(* IEC 61131-3 sources: TA/Tests/RetainTest/OLD/Array test (part 5) *)

    ARRAY_ARRAY_REAL_AUTO[4][0] := ARRAY_ARRAY_REAL_AUTO[4][0] + 1;
    ARRAY_ARRAY_REAL_AUTO[4][1] := ARRAY_ARRAY_REAL_AUTO[4][1] + 1;
    ARRAY_ARRAY_REAL_AUTO[4][2] := ARRAY_ARRAY_REAL_AUTO[4][2] + 1;
    ARRAY_ARRAY_REAL_AUTO[4][3] := ARRAY_ARRAY_REAL_AUTO[4][3] + 1;
    ARRAY_ARRAY_REAL_AUTO[4][4] := ARRAY_ARRAY_REAL_AUTO[4][4] + 1;
    ARRAY_ARRAY_REAL_AUTO[4][5] := ARRAY_ARRAY_REAL_AUTO[4][5] + 1;
    ARRAY_ARRAY_REAL_AUTO[4][6] := ARRAY_ARRAY_REAL_AUTO[4][6] + 1;
    ARRAY_ARRAY_REAL_AUTO[4][7] := ARRAY_ARRAY_REAL_AUTO[4][7] + 1;
    ARRAY_ARRAY_REAL_AUTO[4][8] := ARRAY_ARRAY_REAL_AUTO[4][8] + 1;
    ARRAY_ARRAY_REAL_AUTO[4][9] := ARRAY_ARRAY_REAL_AUTO[4][9] + 1;

    ARRAY_ARRAY_REAL_AUTO[5][0] := ARRAY_ARRAY_REAL_AUTO[5][0] + 1;
    ARRAY_ARRAY_REAL_AUTO[5][1] := ARRAY_ARRAY_REAL_AUTO[5][1] + 1;
    ARRAY_ARRAY_REAL_AUTO[5][2] := ARRAY_ARRAY_REAL_AUTO[5][2] + 1;
    ARRAY_ARRAY_REAL_AUTO[5][3] := ARRAY_ARRAY_REAL_AUTO[5][3] + 1;
    ARRAY_ARRAY_REAL_AUTO[5][4] := ARRAY_ARRAY_REAL_AUTO[5][4] + 1;
    ARRAY_ARRAY_REAL_AUTO[5][5] := ARRAY_ARRAY_REAL_AUTO[5][5] + 1;
    ARRAY_ARRAY_REAL_AUTO[5][6] := ARRAY_ARRAY_REAL_AUTO[5][6] + 1;
    ARRAY_ARRAY_REAL_AUTO[5][7] := ARRAY_ARRAY_REAL_AUTO[5][7] + 1;
    ARRAY_ARRAY_REAL_AUTO[5][8] := ARRAY_ARRAY_REAL_AUTO[5][8] + 1;
    ARRAY_ARRAY_REAL_AUTO[5][9] := ARRAY_ARRAY_REAL_AUTO[5][9] + 1;

    ARRAY_ARRAY_REAL_AUTO[6][0] := ARRAY_ARRAY_REAL_AUTO[6][0] + 1;
    ARRAY_ARRAY_REAL_AUTO[6][1] := ARRAY_ARRAY_REAL_AUTO[6][1] + 1;
    ARRAY_ARRAY_REAL_AUTO[6][2] := ARRAY_ARRAY_REAL_AUTO[6][2] + 1;
    ARRAY_ARRAY_REAL_AUTO[6][3] := ARRAY_ARRAY_REAL_AUTO[6][3] + 1;
    ARRAY_ARRAY_REAL_AUTO[6][4] := ARRAY_ARRAY_REAL_AUTO[6][4] + 1;
    ARRAY_ARRAY_REAL_AUTO[6][5] := ARRAY_ARRAY_REAL_AUTO[6][5] + 1;
    ARRAY_ARRAY_REAL_AUTO[6][6] := ARRAY_ARRAY_REAL_AUTO[6][6] + 1;
    ARRAY_ARRAY_REAL_AUTO[6][7] := ARRAY_ARRAY_REAL_AUTO[6][7] + 1;
    ARRAY_ARRAY_REAL_AUTO[6][8] := ARRAY_ARRAY_REAL_AUTO[6][8] + 1;
    ARRAY_ARRAY_REAL_AUTO[6][9] := ARRAY_ARRAY_REAL_AUTO[6][9] + 1;

    ARRAY_ARRAY_REAL_AUTO[7][0] := ARRAY_ARRAY_REAL_AUTO[6][0];
    ARRAY_ARRAY_REAL_AUTO[7][1] := ARRAY_ARRAY_REAL_AUTO[6][1];
    ARRAY_ARRAY_REAL_AUTO[7][2] := ARRAY_ARRAY_REAL_AUTO[6][2];
    ARRAY_ARRAY_REAL_AUTO[7][3] := ARRAY_ARRAY_REAL_AUTO[6][3];
    ARRAY_ARRAY_REAL_AUTO[7][4] := ARRAY_ARRAY_REAL_AUTO[6][4];
    ARRAY_ARRAY_REAL_AUTO[7][5] := ARRAY_ARRAY_REAL_AUTO[6][5];
    ARRAY_ARRAY_REAL_AUTO[7][6] := ARRAY_ARRAY_REAL_AUTO[6][6];
    ARRAY_ARRAY_REAL_AUTO[7][7] := ARRAY_ARRAY_REAL_AUTO[6][7];
    ARRAY_ARRAY_REAL_AUTO[7][8] := ARRAY_ARRAY_REAL_AUTO[6][8];
    ARRAY_ARRAY_REAL_AUTO[7][9] := ARRAY_ARRAY_REAL_AUTO[6][9];

    ARRAY_ARRAY_SINT_AUTO[0][0] := ARRAY_ARRAY_SINT_AUTO[0][0] + 1;
    ARRAY_ARRAY_SINT_AUTO[0][1] := ARRAY_ARRAY_SINT_AUTO[0][1] + 1;
    ARRAY_ARRAY_SINT_AUTO[0][2] := ARRAY_ARRAY_SINT_AUTO[0][2] + 1;
    ARRAY_ARRAY_SINT_AUTO[0][3] := ARRAY_ARRAY_SINT_AUTO[0][3] + 1;
    ARRAY_ARRAY_SINT_AUTO[0][4] := ARRAY_ARRAY_SINT_AUTO[0][4] + 1;
    ARRAY_ARRAY_SINT_AUTO[0][5] := ARRAY_ARRAY_SINT_AUTO[0][5] + 1;
    ARRAY_ARRAY_SINT_AUTO[0][6] := ARRAY_ARRAY_SINT_AUTO[0][6] + 1;
    ARRAY_ARRAY_SINT_AUTO[0][7] := ARRAY_ARRAY_SINT_AUTO[0][7] + 1;
    ARRAY_ARRAY_SINT_AUTO[0][8] := ARRAY_ARRAY_SINT_AUTO[0][6];
    ARRAY_ARRAY_SINT_AUTO[0][9] := ARRAY_ARRAY_SINT_AUTO[0][7];

    ARRAY_ARRAY_SINT_AUTO[1][0] := ARRAY_ARRAY_SINT_AUTO[1][0] + 1;
    ARRAY_ARRAY_SINT_AUTO[1][1] := ARRAY_ARRAY_SINT_AUTO[1][1] + 1;
    ARRAY_ARRAY_SINT_AUTO[1][2] := ARRAY_ARRAY_SINT_AUTO[1][2] + 1;
    ARRAY_ARRAY_SINT_AUTO[1][3] := ARRAY_ARRAY_SINT_AUTO[1][3] + 1;
    ARRAY_ARRAY_SINT_AUTO[1][4] := ARRAY_ARRAY_SINT_AUTO[1][4] + 1;
    ARRAY_ARRAY_SINT_AUTO[1][5] := ARRAY_ARRAY_SINT_AUTO[1][5] + 1;
    ARRAY_ARRAY_SINT_AUTO[1][6] := ARRAY_ARRAY_SINT_AUTO[1][6] + 1;
    ARRAY_ARRAY_SINT_AUTO[1][7] := ARRAY_ARRAY_SINT_AUTO[1][7] + 1;
    ARRAY_ARRAY_SINT_AUTO[1][8] := ARRAY_ARRAY_SINT_AUTO[1][6];
    ARRAY_ARRAY_SINT_AUTO[1][9] := ARRAY_ARRAY_SINT_AUTO[1][7];

    ARRAY_ARRAY_SINT_AUTO[2][0] := ARRAY_ARRAY_SINT_AUTO[2][0] + 1;
    ARRAY_ARRAY_SINT_AUTO[2][1] := ARRAY_ARRAY_SINT_AUTO[2][1] + 1;
    ARRAY_ARRAY_SINT_AUTO[2][2] := ARRAY_ARRAY_SINT_AUTO[2][2] + 1;
    ARRAY_ARRAY_SINT_AUTO[2][3] := ARRAY_ARRAY_SINT_AUTO[2][3] + 1;
    ARRAY_ARRAY_SINT_AUTO[2][4] := ARRAY_ARRAY_SINT_AUTO[2][4] + 1;
    ARRAY_ARRAY_SINT_AUTO[2][5] := ARRAY_ARRAY_SINT_AUTO[2][5] + 1;
    ARRAY_ARRAY_SINT_AUTO[2][6] := ARRAY_ARRAY_SINT_AUTO[2][6] + 1;
    ARRAY_ARRAY_SINT_AUTO[2][7] := ARRAY_ARRAY_SINT_AUTO[2][7] + 1;
    ARRAY_ARRAY_SINT_AUTO[2][8] := ARRAY_ARRAY_SINT_AUTO[2][8] + 1;
    ARRAY_ARRAY_SINT_AUTO[2][9] := ARRAY_ARRAY_SINT_AUTO[2][9] + 1;

    ARRAY_ARRAY_SINT_AUTO[3][0] := ARRAY_ARRAY_SINT_AUTO[3][0] + 1;
    ARRAY_ARRAY_SINT_AUTO[3][1] := ARRAY_ARRAY_SINT_AUTO[3][1] + 1;
    ARRAY_ARRAY_SINT_AUTO[3][2] := ARRAY_ARRAY_SINT_AUTO[3][2] + 1;
    ARRAY_ARRAY_SINT_AUTO[3][3] := ARRAY_ARRAY_SINT_AUTO[3][3] + 1;
    ARRAY_ARRAY_SINT_AUTO[3][4] := ARRAY_ARRAY_SINT_AUTO[3][4] + 1;
    ARRAY_ARRAY_SINT_AUTO[3][5] := ARRAY_ARRAY_SINT_AUTO[3][5] + 1;
    ARRAY_ARRAY_SINT_AUTO[3][6] := ARRAY_ARRAY_SINT_AUTO[3][6] + 1;
    ARRAY_ARRAY_SINT_AUTO[3][7] := ARRAY_ARRAY_SINT_AUTO[3][7] + 1;
    ARRAY_ARRAY_SINT_AUTO[3][8] := ARRAY_ARRAY_SINT_AUTO[3][8] + 1;
    ARRAY_ARRAY_SINT_AUTO[3][9] := ARRAY_ARRAY_SINT_AUTO[3][9] + 1;

    ARRAY_ARRAY_SINT_AUTO[4][0] := ARRAY_ARRAY_SINT_AUTO[4][0] + 1;
    ARRAY_ARRAY_SINT_AUTO[4][1] := ARRAY_ARRAY_SINT_AUTO[4][1] + 1;
    ARRAY_ARRAY_SINT_AUTO[4][2] := ARRAY_ARRAY_SINT_AUTO[4][2] + 1;
    ARRAY_ARRAY_SINT_AUTO[4][3] := ARRAY_ARRAY_SINT_AUTO[4][3] + 1;
    ARRAY_ARRAY_SINT_AUTO[4][4] := ARRAY_ARRAY_SINT_AUTO[4][4] + 1;
    ARRAY_ARRAY_SINT_AUTO[4][5] := ARRAY_ARRAY_SINT_AUTO[4][5] + 1;
    ARRAY_ARRAY_SINT_AUTO[4][6] := ARRAY_ARRAY_SINT_AUTO[4][6] + 1;
    ARRAY_ARRAY_SINT_AUTO[4][7] := ARRAY_ARRAY_SINT_AUTO[4][7] + 1;
    ARRAY_ARRAY_SINT_AUTO[4][8] := ARRAY_ARRAY_SINT_AUTO[4][8] + 1;
    ARRAY_ARRAY_SINT_AUTO[4][9] := ARRAY_ARRAY_SINT_AUTO[4][9] + 1;

    ARRAY_ARRAY_SINT_AUTO[5][0] := ARRAY_ARRAY_SINT_AUTO[5][0] + 1;
    ARRAY_ARRAY_SINT_AUTO[5][1] := ARRAY_ARRAY_SINT_AUTO[5][1] + 1;
    ARRAY_ARRAY_SINT_AUTO[5][2] := ARRAY_ARRAY_SINT_AUTO[5][2] + 1;
    ARRAY_ARRAY_SINT_AUTO[5][3] := ARRAY_ARRAY_SINT_AUTO[5][3] + 1;
    ARRAY_ARRAY_SINT_AUTO[5][4] := ARRAY_ARRAY_SINT_AUTO[5][4] + 1;
    ARRAY_ARRAY_SINT_AUTO[5][5] := ARRAY_ARRAY_SINT_AUTO[5][5] + 1;
    ARRAY_ARRAY_SINT_AUTO[5][6] := ARRAY_ARRAY_SINT_AUTO[5][6] + 1;
    ARRAY_ARRAY_SINT_AUTO[5][7] := ARRAY_ARRAY_SINT_AUTO[5][7] + 1;
    ARRAY_ARRAY_SINT_AUTO[5][8] := ARRAY_ARRAY_SINT_AUTO[5][8] + 1;
    ARRAY_ARRAY_SINT_AUTO[5][9] := ARRAY_ARRAY_SINT_AUTO[5][9] + 1;

    ARRAY_ARRAY_SINT_AUTO[6][0] := ARRAY_ARRAY_SINT_AUTO[6][0] + 1;
    ARRAY_ARRAY_SINT_AUTO[6][1] := ARRAY_ARRAY_SINT_AUTO[6][1] + 1;
    ARRAY_ARRAY_SINT_AUTO[6][2] := ARRAY_ARRAY_SINT_AUTO[6][2] + 1;
    ARRAY_ARRAY_SINT_AUTO[6][3] := ARRAY_ARRAY_SINT_AUTO[6][3] + 1;
    ARRAY_ARRAY_SINT_AUTO[6][4] := ARRAY_ARRAY_SINT_AUTO[6][4] + 1;
    ARRAY_ARRAY_SINT_AUTO[6][5] := ARRAY_ARRAY_SINT_AUTO[6][5] + 1;
    ARRAY_ARRAY_SINT_AUTO[6][6] := ARRAY_ARRAY_SINT_AUTO[6][6] + 1;
    ARRAY_ARRAY_SINT_AUTO[6][7] := ARRAY_ARRAY_SINT_AUTO[6][7] + 1;
    ARRAY_ARRAY_SINT_AUTO[6][8] := ARRAY_ARRAY_SINT_AUTO[6][8] + 1;
    ARRAY_ARRAY_SINT_AUTO[6][9] := ARRAY_ARRAY_SINT_AUTO[6][9] + 1;

    ARRAY_ARRAY_SINT_AUTO[7][0] := ARRAY_ARRAY_SINT_AUTO[6][0];
    ARRAY_ARRAY_SINT_AUTO[7][1] := ARRAY_ARRAY_SINT_AUTO[6][1];
    ARRAY_ARRAY_SINT_AUTO[7][2] := ARRAY_ARRAY_SINT_AUTO[6][2];
    ARRAY_ARRAY_SINT_AUTO[7][3] := ARRAY_ARRAY_SINT_AUTO[6][3];
    ARRAY_ARRAY_SINT_AUTO[7][4] := ARRAY_ARRAY_SINT_AUTO[6][4];
    ARRAY_ARRAY_SINT_AUTO[7][5] := ARRAY_ARRAY_SINT_AUTO[6][5];
    ARRAY_ARRAY_SINT_AUTO[7][6] := ARRAY_ARRAY_SINT_AUTO[6][6];
    ARRAY_ARRAY_SINT_AUTO[7][7] := ARRAY_ARRAY_SINT_AUTO[6][7];
    ARRAY_ARRAY_SINT_AUTO[7][8] := ARRAY_ARRAY_SINT_AUTO[6][8];
    ARRAY_ARRAY_SINT_AUTO[7][9] := ARRAY_ARRAY_SINT_AUTO[6][9];

    ARRAY_ARRAY_STRING_AUTO[0][0] := ANY_TO_STRING(ARRAY_ARRAY_DINT_AUTO[0][0]) + ' ' + ANY_TO_STRING(ARRAY_ARRAY_TIME_AUTO[0][0]);
    ARRAY_ARRAY_STRING_AUTO[0][1] := ANY_TO_STRING(ARRAY_ARRAY_DINT_AUTO[0][1]) + ' ' + ANY_TO_STRING(ARRAY_ARRAY_TIME_AUTO[0][1]);
    ARRAY_ARRAY_STRING_AUTO[0][2] := ANY_TO_STRING(ARRAY_ARRAY_DINT_AUTO[0][2]) + ' ' + ANY_TO_STRING(ARRAY_ARRAY_TIME_AUTO[0][2]);
    ARRAY_ARRAY_STRING_AUTO[0][3] := ANY_TO_STRING(ARRAY_ARRAY_DINT_AUTO[0][3]) + ' ' + ANY_TO_STRING(ARRAY_ARRAY_TIME_AUTO[0][3]);
    ARRAY_ARRAY_STRING_AUTO[0][4] := ANY_TO_STRING(ARRAY_ARRAY_DINT_AUTO[0][4]) + ' ' + ANY_TO_STRING(ARRAY_ARRAY_TIME_AUTO[0][4]);
    ARRAY_ARRAY_STRING_AUTO[0][5] := ANY_TO_STRING(ARRAY_ARRAY_DINT_AUTO[0][5]) + ' ' + ANY_TO_STRING(ARRAY_ARRAY_TIME_AUTO[0][5]);
    ARRAY_ARRAY_STRING_AUTO[0][6] := ANY_TO_STRING(ARRAY_ARRAY_DINT_AUTO[0][6]) + ' ' + ANY_TO_STRING(ARRAY_ARRAY_TIME_AUTO[0][6]);
    ARRAY_ARRAY_STRING_AUTO[0][7] := ANY_TO_STRING(ARRAY_ARRAY_DINT_AUTO[0][7]) + ' ' + ANY_TO_STRING(ARRAY_ARRAY_TIME_AUTO[0][7]);
    ARRAY_ARRAY_STRING_AUTO[0][8] := ARRAY_ARRAY_STRING_AUTO[0][6];
    ARRAY_ARRAY_STRING_AUTO[0][9] := ARRAY_ARRAY_STRING_AUTO[0][7];

    ARRAY_ARRAY_STRING_AUTO[1][0] := ANY_TO_STRING(ARRAY_ARRAY_DINT_AUTO[1][0]) + ' ' + ANY_TO_STRING(ARRAY_ARRAY_TIME_AUTO[1][0]);
    ARRAY_ARRAY_STRING_AUTO[1][1] := ANY_TO_STRING(ARRAY_ARRAY_DINT_AUTO[1][1]) + ' ' + ANY_TO_STRING(ARRAY_ARRAY_TIME_AUTO[1][1]);
    ARRAY_ARRAY_STRING_AUTO[1][2] := ANY_TO_STRING(ARRAY_ARRAY_DINT_AUTO[1][2]) + ' ' + ANY_TO_STRING(ARRAY_ARRAY_TIME_AUTO[1][2]);
    ARRAY_ARRAY_STRING_AUTO[1][3] := ANY_TO_STRING(ARRAY_ARRAY_DINT_AUTO[1][3]) + ' ' + ANY_TO_STRING(ARRAY_ARRAY_TIME_AUTO[1][3]);
    ARRAY_ARRAY_STRING_AUTO[1][4] := ANY_TO_STRING(ARRAY_ARRAY_DINT_AUTO[1][4]) + ' ' + ANY_TO_STRING(ARRAY_ARRAY_TIME_AUTO[1][4]);
    ARRAY_ARRAY_STRING_AUTO[1][5] := ANY_TO_STRING(ARRAY_ARRAY_DINT_AUTO[1][5]) + ' ' + ANY_TO_STRING(ARRAY_ARRAY_TIME_AUTO[1][5]);
    ARRAY_ARRAY_STRING_AUTO[1][6] := ANY_TO_STRING(ARRAY_ARRAY_DINT_AUTO[1][6]) + ' ' + ANY_TO_STRING(ARRAY_ARRAY_TIME_AUTO[1][6]);
    ARRAY_ARRAY_STRING_AUTO[1][7] := ANY_TO_STRING(ARRAY_ARRAY_DINT_AUTO[1][7]) + ' ' + ANY_TO_STRING(ARRAY_ARRAY_TIME_AUTO[1][7]);
    ARRAY_ARRAY_STRING_AUTO[1][8] := ARRAY_ARRAY_STRING_AUTO[1][6];
    ARRAY_ARRAY_STRING_AUTO[1][9] := ARRAY_ARRAY_STRING_AUTO[1][7];

    ARRAY_ARRAY_STRING_AUTO[2][0] := ANY_TO_STRING(ARRAY_ARRAY_DINT_AUTO[2][0]) + ' ' + ANY_TO_STRING(ARRAY_ARRAY_TIME_AUTO[2][0]);
    ARRAY_ARRAY_STRING_AUTO[2][1] := ANY_TO_STRING(ARRAY_ARRAY_DINT_AUTO[2][1]) + ' ' + ANY_TO_STRING(ARRAY_ARRAY_TIME_AUTO[2][1]);
    ARRAY_ARRAY_STRING_AUTO[2][2] := ANY_TO_STRING(ARRAY_ARRAY_DINT_AUTO[2][2]) + ' ' + ANY_TO_STRING(ARRAY_ARRAY_TIME_AUTO[2][2]);
    ARRAY_ARRAY_STRING_AUTO[2][3] := ANY_TO_STRING(ARRAY_ARRAY_DINT_AUTO[2][3]) + ' ' + ANY_TO_STRING(ARRAY_ARRAY_TIME_AUTO[2][3]);
    ARRAY_ARRAY_STRING_AUTO[2][4] := ANY_TO_STRING(ARRAY_ARRAY_DINT_AUTO[2][4]) + ' ' + ANY_TO_STRING(ARRAY_ARRAY_TIME_AUTO[2][4]);
    ARRAY_ARRAY_STRING_AUTO[2][5] := ANY_TO_STRING(ARRAY_ARRAY_DINT_AUTO[2][5]) + ' ' + ANY_TO_STRING(ARRAY_ARRAY_TIME_AUTO[2][5]);
    ARRAY_ARRAY_STRING_AUTO[2][6] := ANY_TO_STRING(ARRAY_ARRAY_DINT_AUTO[2][6]) + ' ' + ANY_TO_STRING(ARRAY_ARRAY_TIME_AUTO[2][6]);
    ARRAY_ARRAY_STRING_AUTO[2][7] := ANY_TO_STRING(ARRAY_ARRAY_DINT_AUTO[2][7]) + ' ' + ANY_TO_STRING(ARRAY_ARRAY_TIME_AUTO[2][7]);
    ARRAY_ARRAY_STRING_AUTO[2][8] := ANY_TO_STRING(ARRAY_ARRAY_DINT_AUTO[2][8]) + ' ' + ANY_TO_STRING(ARRAY_ARRAY_TIME_AUTO[2][8]);
    ARRAY_ARRAY_STRING_AUTO[2][9] := ANY_TO_STRING(ARRAY_ARRAY_DINT_AUTO[2][9]) + ' ' + ANY_TO_STRING(ARRAY_ARRAY_TIME_AUTO[2][9]);

    ARRAY_ARRAY_STRING_AUTO[3][0] := ANY_TO_STRING(ARRAY_ARRAY_DINT_AUTO[3][0]) + ' ' + ANY_TO_STRING(ARRAY_ARRAY_TIME_AUTO[3][0]);
    ARRAY_ARRAY_STRING_AUTO[3][1] := ANY_TO_STRING(ARRAY_ARRAY_DINT_AUTO[3][1]) + ' ' + ANY_TO_STRING(ARRAY_ARRAY_TIME_AUTO[3][1]);
    ARRAY_ARRAY_STRING_AUTO[3][2] := ANY_TO_STRING(ARRAY_ARRAY_DINT_AUTO[3][2]) + ' ' + ANY_TO_STRING(ARRAY_ARRAY_TIME_AUTO[3][2]);
    ARRAY_ARRAY_STRING_AUTO[3][3] := ANY_TO_STRING(ARRAY_ARRAY_DINT_AUTO[3][3]) + ' ' + ANY_TO_STRING(ARRAY_ARRAY_TIME_AUTO[3][3]);
    ARRAY_ARRAY_STRING_AUTO[3][4] := ANY_TO_STRING(ARRAY_ARRAY_DINT_AUTO[3][4]) + ' ' + ANY_TO_STRING(ARRAY_ARRAY_TIME_AUTO[3][4]);
    ARRAY_ARRAY_STRING_AUTO[3][5] := ANY_TO_STRING(ARRAY_ARRAY_DINT_AUTO[3][5]) + ' ' + ANY_TO_STRING(ARRAY_ARRAY_TIME_AUTO[3][5]);
    ARRAY_ARRAY_STRING_AUTO[3][6] := ANY_TO_STRING(ARRAY_ARRAY_DINT_AUTO[3][6]) + ' ' + ANY_TO_STRING(ARRAY_ARRAY_TIME_AUTO[3][6]);
    ARRAY_ARRAY_STRING_AUTO[3][7] := ANY_TO_STRING(ARRAY_ARRAY_DINT_AUTO[3][7]) + ' ' + ANY_TO_STRING(ARRAY_ARRAY_TIME_AUTO[3][7]);
    ARRAY_ARRAY_STRING_AUTO[3][8] := ANY_TO_STRING(ARRAY_ARRAY_DINT_AUTO[3][8]) + ' ' + ANY_TO_STRING(ARRAY_ARRAY_TIME_AUTO[3][8]);
    ARRAY_ARRAY_STRING_AUTO[3][9] := ANY_TO_STRING(ARRAY_ARRAY_DINT_AUTO[3][9]) + ' ' + ANY_TO_STRING(ARRAY_ARRAY_TIME_AUTO[3][9]);

    ARRAY_ARRAY_STRING_AUTO[4][0] := ANY_TO_STRING(ARRAY_ARRAY_DINT_AUTO[4][0]) + ' ' + ANY_TO_STRING(ARRAY_ARRAY_TIME_AUTO[4][0]);
    ARRAY_ARRAY_STRING_AUTO[4][1] := ANY_TO_STRING(ARRAY_ARRAY_DINT_AUTO[4][1]) + ' ' + ANY_TO_STRING(ARRAY_ARRAY_TIME_AUTO[4][1]);
    ARRAY_ARRAY_STRING_AUTO[4][2] := ANY_TO_STRING(ARRAY_ARRAY_DINT_AUTO[4][2]) + ' ' + ANY_TO_STRING(ARRAY_ARRAY_TIME_AUTO[4][2]);
    ARRAY_ARRAY_STRING_AUTO[4][3] := ANY_TO_STRING(ARRAY_ARRAY_DINT_AUTO[4][3]) + ' ' + ANY_TO_STRING(ARRAY_ARRAY_TIME_AUTO[4][3]);
    ARRAY_ARRAY_STRING_AUTO[4][4] := ANY_TO_STRING(ARRAY_ARRAY_DINT_AUTO[4][4]) + ' ' + ANY_TO_STRING(ARRAY_ARRAY_TIME_AUTO[4][4]);
    ARRAY_ARRAY_STRING_AUTO[4][5] := ANY_TO_STRING(ARRAY_ARRAY_DINT_AUTO[4][5]) + ' ' + ANY_TO_STRING(ARRAY_ARRAY_TIME_AUTO[4][5]);
    ARRAY_ARRAY_STRING_AUTO[4][6] := ANY_TO_STRING(ARRAY_ARRAY_DINT_AUTO[4][6]) + ' ' + ANY_TO_STRING(ARRAY_ARRAY_TIME_AUTO[4][6]);
    ARRAY_ARRAY_STRING_AUTO[4][7] := ANY_TO_STRING(ARRAY_ARRAY_DINT_AUTO[4][7]) + ' ' + ANY_TO_STRING(ARRAY_ARRAY_TIME_AUTO[4][7]);
    ARRAY_ARRAY_STRING_AUTO[4][8] := ANY_TO_STRING(ARRAY_ARRAY_DINT_AUTO[4][8]) + ' ' + ANY_TO_STRING(ARRAY_ARRAY_TIME_AUTO[4][8]);
    ARRAY_ARRAY_STRING_AUTO[4][9] := ANY_TO_STRING(ARRAY_ARRAY_DINT_AUTO[4][9]) + ' ' + ANY_TO_STRING(ARRAY_ARRAY_TIME_AUTO[4][9]);

    ARRAY_ARRAY_STRING_AUTO[5][0] := ANY_TO_STRING(ARRAY_ARRAY_DINT_AUTO[5][0]) + ' ' + ANY_TO_STRING(ARRAY_ARRAY_TIME_AUTO[5][0]);
    ARRAY_ARRAY_STRING_AUTO[5][1] := ANY_TO_STRING(ARRAY_ARRAY_DINT_AUTO[5][1]) + ' ' + ANY_TO_STRING(ARRAY_ARRAY_TIME_AUTO[5][1]);
    ARRAY_ARRAY_STRING_AUTO[5][2] := ANY_TO_STRING(ARRAY_ARRAY_DINT_AUTO[5][2]) + ' ' + ANY_TO_STRING(ARRAY_ARRAY_TIME_AUTO[5][2]);
    ARRAY_ARRAY_STRING_AUTO[5][3] := ANY_TO_STRING(ARRAY_ARRAY_DINT_AUTO[5][3]) + ' ' + ANY_TO_STRING(ARRAY_ARRAY_TIME_AUTO[5][3]);
    ARRAY_ARRAY_STRING_AUTO[5][4] := ANY_TO_STRING(ARRAY_ARRAY_DINT_AUTO[5][4]) + ' ' + ANY_TO_STRING(ARRAY_ARRAY_TIME_AUTO[5][4]);
    ARRAY_ARRAY_STRING_AUTO[5][5] := ANY_TO_STRING(ARRAY_ARRAY_DINT_AUTO[5][5]) + ' ' + ANY_TO_STRING(ARRAY_ARRAY_TIME_AUTO[5][5]);
    ARRAY_ARRAY_STRING_AUTO[5][6] := ANY_TO_STRING(ARRAY_ARRAY_DINT_AUTO[5][6]) + ' ' + ANY_TO_STRING(ARRAY_ARRAY_TIME_AUTO[5][6]);
    ARRAY_ARRAY_STRING_AUTO[5][7] := ANY_TO_STRING(ARRAY_ARRAY_DINT_AUTO[5][7]) + ' ' + ANY_TO_STRING(ARRAY_ARRAY_TIME_AUTO[5][7]);
    ARRAY_ARRAY_STRING_AUTO[5][8] := ANY_TO_STRING(ARRAY_ARRAY_DINT_AUTO[5][8]) + ' ' + ANY_TO_STRING(ARRAY_ARRAY_TIME_AUTO[5][8]);
    ARRAY_ARRAY_STRING_AUTO[5][9] := ANY_TO_STRING(ARRAY_ARRAY_DINT_AUTO[5][9]) + ' ' + ANY_TO_STRING(ARRAY_ARRAY_TIME_AUTO[5][9]);

    ARRAY_ARRAY_STRING_AUTO[6][0] := ANY_TO_STRING(ARRAY_ARRAY_DINT_AUTO[6][0]) + ' ' + ANY_TO_STRING(ARRAY_ARRAY_TIME_AUTO[6][0]);
    ARRAY_ARRAY_STRING_AUTO[6][1] := ANY_TO_STRING(ARRAY_ARRAY_DINT_AUTO[6][1]) + ' ' + ANY_TO_STRING(ARRAY_ARRAY_TIME_AUTO[6][1]);
    ARRAY_ARRAY_STRING_AUTO[6][2] := ANY_TO_STRING(ARRAY_ARRAY_DINT_AUTO[6][2]) + ' ' + ANY_TO_STRING(ARRAY_ARRAY_TIME_AUTO[6][2]);
    ARRAY_ARRAY_STRING_AUTO[6][3] := ANY_TO_STRING(ARRAY_ARRAY_DINT_AUTO[6][3]) + ' ' + ANY_TO_STRING(ARRAY_ARRAY_TIME_AUTO[6][3]);
    ARRAY_ARRAY_STRING_AUTO[6][4] := ANY_TO_STRING(ARRAY_ARRAY_DINT_AUTO[6][4]) + ' ' + ANY_TO_STRING(ARRAY_ARRAY_TIME_AUTO[6][4]);
    ARRAY_ARRAY_STRING_AUTO[6][5] := ANY_TO_STRING(ARRAY_ARRAY_DINT_AUTO[6][5]) + ' ' + ANY_TO_STRING(ARRAY_ARRAY_TIME_AUTO[6][5]);
    ARRAY_ARRAY_STRING_AUTO[6][6] := ANY_TO_STRING(ARRAY_ARRAY_DINT_AUTO[6][6]) + ' ' + ANY_TO_STRING(ARRAY_ARRAY_TIME_AUTO[6][6]);
    ARRAY_ARRAY_STRING_AUTO[6][7] := ANY_TO_STRING(ARRAY_ARRAY_DINT_AUTO[6][7]) + ' ' + ANY_TO_STRING(ARRAY_ARRAY_TIME_AUTO[6][7]);
    ARRAY_ARRAY_STRING_AUTO[6][8] := ANY_TO_STRING(ARRAY_ARRAY_DINT_AUTO[6][8]) + ' ' + ANY_TO_STRING(ARRAY_ARRAY_TIME_AUTO[6][8]);
    ARRAY_ARRAY_STRING_AUTO[6][9] := ANY_TO_STRING(ARRAY_ARRAY_DINT_AUTO[6][9]) + ' ' + ANY_TO_STRING(ARRAY_ARRAY_TIME_AUTO[6][9]);

    ARRAY_ARRAY_STRING_AUTO[7][0] := ARRAY_ARRAY_STRING_AUTO[6][0];
    ARRAY_ARRAY_STRING_AUTO[7][1] := ARRAY_ARRAY_STRING_AUTO[6][1];
    ARRAY_ARRAY_STRING_AUTO[7][2] := ARRAY_ARRAY_STRING_AUTO[6][2];
    ARRAY_ARRAY_STRING_AUTO[7][3] := ARRAY_ARRAY_STRING_AUTO[6][3];
    ARRAY_ARRAY_STRING_AUTO[7][4] := ARRAY_ARRAY_STRING_AUTO[6][4];
    ARRAY_ARRAY_STRING_AUTO[7][5] := ARRAY_ARRAY_STRING_AUTO[6][5];
    ARRAY_ARRAY_STRING_AUTO[7][6] := ARRAY_ARRAY_STRING_AUTO[6][6];
    ARRAY_ARRAY_STRING_AUTO[7][7] := ARRAY_ARRAY_STRING_AUTO[6][7];
    ARRAY_ARRAY_STRING_AUTO[7][8] := ARRAY_ARRAY_STRING_AUTO[6][8];
    ARRAY_ARRAY_STRING_AUTO[7][9] := ARRAY_ARRAY_STRING_AUTO[6][9];

    ARRAY_ARRAY_TIME_AUTO[0][0] := ARRAY_ARRAY_TIME_AUTO[0][0] + PULSE_TIME;
    ARRAY_ARRAY_TIME_AUTO[0][1] := ARRAY_ARRAY_TIME_AUTO[0][1] + PULSE_TIME;
    ARRAY_ARRAY_TIME_AUTO[0][2] := ARRAY_ARRAY_TIME_AUTO[0][2] + PULSE_TIME;
    ARRAY_ARRAY_TIME_AUTO[0][3] := ARRAY_ARRAY_TIME_AUTO[0][3] + PULSE_TIME;
    ARRAY_ARRAY_TIME_AUTO[0][4] := ARRAY_ARRAY_TIME_AUTO[0][4] + PULSE_TIME;
    ARRAY_ARRAY_TIME_AUTO[0][5] := ARRAY_ARRAY_TIME_AUTO[0][5] + PULSE_TIME;
    ARRAY_ARRAY_TIME_AUTO[0][6] := ARRAY_ARRAY_TIME_AUTO[0][6] + PULSE_TIME;
    ARRAY_ARRAY_TIME_AUTO[0][7] := ARRAY_ARRAY_TIME_AUTO[0][7] + PULSE_TIME;
    ARRAY_ARRAY_TIME_AUTO[0][8] := ARRAY_ARRAY_TIME_AUTO[0][6];
    ARRAY_ARRAY_TIME_AUTO[0][9] := ARRAY_ARRAY_TIME_AUTO[0][7];

    ARRAY_ARRAY_TIME_AUTO[1][0] := ARRAY_ARRAY_TIME_AUTO[1][0] + PULSE_TIME;
    ARRAY_ARRAY_TIME_AUTO[1][1] := ARRAY_ARRAY_TIME_AUTO[1][1] + PULSE_TIME;
    ARRAY_ARRAY_TIME_AUTO[1][2] := ARRAY_ARRAY_TIME_AUTO[1][2] + PULSE_TIME;
    ARRAY_ARRAY_TIME_AUTO[1][3] := ARRAY_ARRAY_TIME_AUTO[1][3] + PULSE_TIME;
    ARRAY_ARRAY_TIME_AUTO[1][4] := ARRAY_ARRAY_TIME_AUTO[1][4] + PULSE_TIME;
    ARRAY_ARRAY_TIME_AUTO[1][5] := ARRAY_ARRAY_TIME_AUTO[1][5] + PULSE_TIME;
    ARRAY_ARRAY_TIME_AUTO[1][6] := ARRAY_ARRAY_TIME_AUTO[1][6] + PULSE_TIME;
    ARRAY_ARRAY_TIME_AUTO[1][7] := ARRAY_ARRAY_TIME_AUTO[1][7] + PULSE_TIME;
    ARRAY_ARRAY_TIME_AUTO[1][8] := ARRAY_ARRAY_TIME_AUTO[1][6];
    ARRAY_ARRAY_TIME_AUTO[1][9] := ARRAY_ARRAY_TIME_AUTO[1][7];

    ARRAY_ARRAY_TIME_AUTO[2][0] := ARRAY_ARRAY_TIME_AUTO[2][0] + PULSE_TIME;
    ARRAY_ARRAY_TIME_AUTO[2][1] := ARRAY_ARRAY_TIME_AUTO[2][1] + PULSE_TIME;
    ARRAY_ARRAY_TIME_AUTO[2][2] := ARRAY_ARRAY_TIME_AUTO[2][2] + PULSE_TIME;
    ARRAY_ARRAY_TIME_AUTO[2][3] := ARRAY_ARRAY_TIME_AUTO[2][3] + PULSE_TIME;
    ARRAY_ARRAY_TIME_AUTO[2][4] := ARRAY_ARRAY_TIME_AUTO[2][4] + PULSE_TIME;
    ARRAY_ARRAY_TIME_AUTO[2][5] := ARRAY_ARRAY_TIME_AUTO[2][5] + PULSE_TIME;
    ARRAY_ARRAY_TIME_AUTO[2][6] := ARRAY_ARRAY_TIME_AUTO[2][6] + PULSE_TIME;
    ARRAY_ARRAY_TIME_AUTO[2][7] := ARRAY_ARRAY_TIME_AUTO[2][7] + PULSE_TIME;
    ARRAY_ARRAY_TIME_AUTO[2][8] := ARRAY_ARRAY_TIME_AUTO[2][8] + PULSE_TIME;
    ARRAY_ARRAY_TIME_AUTO[2][9] := ARRAY_ARRAY_TIME_AUTO[2][9] + PULSE_TIME;

    ARRAY_ARRAY_TIME_AUTO[3][0] := ARRAY_ARRAY_TIME_AUTO[3][0] + PULSE_TIME;
    ARRAY_ARRAY_TIME_AUTO[3][1] := ARRAY_ARRAY_TIME_AUTO[3][1] + PULSE_TIME;
    ARRAY_ARRAY_TIME_AUTO[3][2] := ARRAY_ARRAY_TIME_AUTO[3][2] + PULSE_TIME;
    ARRAY_ARRAY_TIME_AUTO[3][3] := ARRAY_ARRAY_TIME_AUTO[3][3] + PULSE_TIME;
    ARRAY_ARRAY_TIME_AUTO[3][4] := ARRAY_ARRAY_TIME_AUTO[3][4] + PULSE_TIME;
    ARRAY_ARRAY_TIME_AUTO[3][5] := ARRAY_ARRAY_TIME_AUTO[3][5] + PULSE_TIME;
    ARRAY_ARRAY_TIME_AUTO[3][6] := ARRAY_ARRAY_TIME_AUTO[3][6] + PULSE_TIME;
    ARRAY_ARRAY_TIME_AUTO[3][7] := ARRAY_ARRAY_TIME_AUTO[3][7] + PULSE_TIME;
    ARRAY_ARRAY_TIME_AUTO[3][8] := ARRAY_ARRAY_TIME_AUTO[3][8] + PULSE_TIME;
    ARRAY_ARRAY_TIME_AUTO[3][9] := ARRAY_ARRAY_TIME_AUTO[3][9] + PULSE_TIME;

    ARRAY_ARRAY_TIME_AUTO[4][0] := ARRAY_ARRAY_TIME_AUTO[4][0] + PULSE_TIME;
    ARRAY_ARRAY_TIME_AUTO[4][1] := ARRAY_ARRAY_TIME_AUTO[4][1] + PULSE_TIME;
    ARRAY_ARRAY_TIME_AUTO[4][2] := ARRAY_ARRAY_TIME_AUTO[4][2] + PULSE_TIME;
    ARRAY_ARRAY_TIME_AUTO[4][3] := ARRAY_ARRAY_TIME_AUTO[4][3] + PULSE_TIME;
    ARRAY_ARRAY_TIME_AUTO[4][4] := ARRAY_ARRAY_TIME_AUTO[4][4] + PULSE_TIME;
    ARRAY_ARRAY_TIME_AUTO[4][5] := ARRAY_ARRAY_TIME_AUTO[4][5] + PULSE_TIME;
    ARRAY_ARRAY_TIME_AUTO[4][6] := ARRAY_ARRAY_TIME_AUTO[4][6] + PULSE_TIME;
    ARRAY_ARRAY_TIME_AUTO[4][7] := ARRAY_ARRAY_TIME_AUTO[4][7] + PULSE_TIME;
    ARRAY_ARRAY_TIME_AUTO[4][8] := ARRAY_ARRAY_TIME_AUTO[4][8] + PULSE_TIME;
    ARRAY_ARRAY_TIME_AUTO[4][9] := ARRAY_ARRAY_TIME_AUTO[4][9] + PULSE_TIME;

    ARRAY_ARRAY_TIME_AUTO[5][0] := ARRAY_ARRAY_TIME_AUTO[5][0] + PULSE_TIME;
    ARRAY_ARRAY_TIME_AUTO[5][1] := ARRAY_ARRAY_TIME_AUTO[5][1] + PULSE_TIME;
    ARRAY_ARRAY_TIME_AUTO[5][2] := ARRAY_ARRAY_TIME_AUTO[5][2] + PULSE_TIME;
    ARRAY_ARRAY_TIME_AUTO[5][3] := ARRAY_ARRAY_TIME_AUTO[5][3] + PULSE_TIME;
    ARRAY_ARRAY_TIME_AUTO[5][4] := ARRAY_ARRAY_TIME_AUTO[5][4] + PULSE_TIME;
    ARRAY_ARRAY_TIME_AUTO[5][5] := ARRAY_ARRAY_TIME_AUTO[5][5] + PULSE_TIME;
    ARRAY_ARRAY_TIME_AUTO[5][6] := ARRAY_ARRAY_TIME_AUTO[5][6] + PULSE_TIME;
    ARRAY_ARRAY_TIME_AUTO[5][7] := ARRAY_ARRAY_TIME_AUTO[5][7] + PULSE_TIME;
    ARRAY_ARRAY_TIME_AUTO[5][8] := ARRAY_ARRAY_TIME_AUTO[5][8] + PULSE_TIME;
    ARRAY_ARRAY_TIME_AUTO[5][9] := ARRAY_ARRAY_TIME_AUTO[5][9] + PULSE_TIME;

    ARRAY_ARRAY_TIME_AUTO[6][0] := ARRAY_ARRAY_TIME_AUTO[6][0] + PULSE_TIME;
    ARRAY_ARRAY_TIME_AUTO[6][1] := ARRAY_ARRAY_TIME_AUTO[6][1] + PULSE_TIME;
    ARRAY_ARRAY_TIME_AUTO[6][2] := ARRAY_ARRAY_TIME_AUTO[6][2] + PULSE_TIME;
    ARRAY_ARRAY_TIME_AUTO[6][3] := ARRAY_ARRAY_TIME_AUTO[6][3] + PULSE_TIME;
    ARRAY_ARRAY_TIME_AUTO[6][4] := ARRAY_ARRAY_TIME_AUTO[6][4] + PULSE_TIME;
    ARRAY_ARRAY_TIME_AUTO[6][5] := ARRAY_ARRAY_TIME_AUTO[6][5] + PULSE_TIME;
    ARRAY_ARRAY_TIME_AUTO[6][6] := ARRAY_ARRAY_TIME_AUTO[6][6] + PULSE_TIME;
    ARRAY_ARRAY_TIME_AUTO[6][7] := ARRAY_ARRAY_TIME_AUTO[6][7] + PULSE_TIME;
    ARRAY_ARRAY_TIME_AUTO[6][8] := ARRAY_ARRAY_TIME_AUTO[6][8] + PULSE_TIME;
    ARRAY_ARRAY_TIME_AUTO[6][9] := ARRAY_ARRAY_TIME_AUTO[6][9] + PULSE_TIME;

    ARRAY_ARRAY_TIME_AUTO[7][0] := ARRAY_ARRAY_TIME_AUTO[6][0];
    ARRAY_ARRAY_TIME_AUTO[7][1] := ARRAY_ARRAY_TIME_AUTO[6][1];
    ARRAY_ARRAY_TIME_AUTO[7][2] := ARRAY_ARRAY_TIME_AUTO[6][2];
    ARRAY_ARRAY_TIME_AUTO[7][3] := ARRAY_ARRAY_TIME_AUTO[6][3];
    ARRAY_ARRAY_TIME_AUTO[7][4] := ARRAY_ARRAY_TIME_AUTO[6][4];
    ARRAY_ARRAY_TIME_AUTO[7][5] := ARRAY_ARRAY_TIME_AUTO[6][5];
    ARRAY_ARRAY_TIME_AUTO[7][6] := ARRAY_ARRAY_TIME_AUTO[6][6];
    ARRAY_ARRAY_TIME_AUTO[7][7] := ARRAY_ARRAY_TIME_AUTO[6][7];
    ARRAY_ARRAY_TIME_AUTO[7][8] := ARRAY_ARRAY_TIME_AUTO[6][6];
    ARRAY_ARRAY_TIME_AUTO[7][9] := ARRAY_ARRAY_TIME_AUTO[6][7];

    ARRAY_ARRAY_UDINT_AUTO[0][0] := ARRAY_ARRAY_UDINT_AUTO[0][0] + 1;
    ARRAY_ARRAY_UDINT_AUTO[0][1] := ARRAY_ARRAY_UDINT_AUTO[0][1] + 1;
    ARRAY_ARRAY_UDINT_AUTO[0][2] := ARRAY_ARRAY_UDINT_AUTO[0][2] + 1;
    ARRAY_ARRAY_UDINT_AUTO[0][3] := ARRAY_ARRAY_UDINT_AUTO[0][3] + 1;
    ARRAY_ARRAY_UDINT_AUTO[0][4] := ARRAY_ARRAY_UDINT_AUTO[0][4] + 1;
    ARRAY_ARRAY_UDINT_AUTO[0][5] := ARRAY_ARRAY_UDINT_AUTO[0][5] + 1;
    ARRAY_ARRAY_UDINT_AUTO[0][6] := ARRAY_ARRAY_UDINT_AUTO[0][6] + 1;
    ARRAY_ARRAY_UDINT_AUTO[0][7] := ARRAY_ARRAY_UDINT_AUTO[0][7] + 1;
    ARRAY_ARRAY_UDINT_AUTO[0][8] := ARRAY_ARRAY_UDINT_AUTO[0][6];
    ARRAY_ARRAY_UDINT_AUTO[0][9] := ARRAY_ARRAY_UDINT_AUTO[0][7];

    ARRAY_ARRAY_UDINT_AUTO[1][0] := ARRAY_ARRAY_UDINT_AUTO[1][0] + 1;
    ARRAY_ARRAY_UDINT_AUTO[1][1] := ARRAY_ARRAY_UDINT_AUTO[1][1] + 1;
    ARRAY_ARRAY_UDINT_AUTO[1][2] := ARRAY_ARRAY_UDINT_AUTO[1][2] + 1;
    ARRAY_ARRAY_UDINT_AUTO[1][3] := ARRAY_ARRAY_UDINT_AUTO[1][3] + 1;
    ARRAY_ARRAY_UDINT_AUTO[1][4] := ARRAY_ARRAY_UDINT_AUTO[1][4] + 1;
    ARRAY_ARRAY_UDINT_AUTO[1][5] := ARRAY_ARRAY_UDINT_AUTO[1][5] + 1;
    ARRAY_ARRAY_UDINT_AUTO[1][6] := ARRAY_ARRAY_UDINT_AUTO[1][6] + 1;
    ARRAY_ARRAY_UDINT_AUTO[1][7] := ARRAY_ARRAY_UDINT_AUTO[1][7] + 1;
    ARRAY_ARRAY_UDINT_AUTO[1][8] := ARRAY_ARRAY_UDINT_AUTO[1][6];
    ARRAY_ARRAY_UDINT_AUTO[1][9] := ARRAY_ARRAY_UDINT_AUTO[1][7];

    ARRAY_ARRAY_UDINT_AUTO[2][0] := ARRAY_ARRAY_UDINT_AUTO[2][0] + 1;
    ARRAY_ARRAY_UDINT_AUTO[2][1] := ARRAY_ARRAY_UDINT_AUTO[2][1] + 1;
    ARRAY_ARRAY_UDINT_AUTO[2][2] := ARRAY_ARRAY_UDINT_AUTO[2][2] + 1;
    ARRAY_ARRAY_UDINT_AUTO[2][3] := ARRAY_ARRAY_UDINT_AUTO[2][3] + 1;
    ARRAY_ARRAY_UDINT_AUTO[2][4] := ARRAY_ARRAY_UDINT_AUTO[2][4] + 1;
    ARRAY_ARRAY_UDINT_AUTO[2][5] := ARRAY_ARRAY_UDINT_AUTO[2][5] + 1;
    ARRAY_ARRAY_UDINT_AUTO[2][6] := ARRAY_ARRAY_UDINT_AUTO[2][6] + 1;
    ARRAY_ARRAY_UDINT_AUTO[2][7] := ARRAY_ARRAY_UDINT_AUTO[2][7] + 1;
    ARRAY_ARRAY_UDINT_AUTO[2][8] := ARRAY_ARRAY_UDINT_AUTO[2][8] + 1;
    ARRAY_ARRAY_UDINT_AUTO[2][9] := ARRAY_ARRAY_UDINT_AUTO[2][9] + 1;

    ARRAY_ARRAY_UDINT_AUTO[3][0] := ARRAY_ARRAY_UDINT_AUTO[3][0] + 1;
    ARRAY_ARRAY_UDINT_AUTO[3][1] := ARRAY_ARRAY_UDINT_AUTO[3][1] + 1;
    ARRAY_ARRAY_UDINT_AUTO[3][2] := ARRAY_ARRAY_UDINT_AUTO[3][2] + 1;
    ARRAY_ARRAY_UDINT_AUTO[3][3] := ARRAY_ARRAY_UDINT_AUTO[3][3] + 1;
    ARRAY_ARRAY_UDINT_AUTO[3][4] := ARRAY_ARRAY_UDINT_AUTO[3][4] + 1;
    ARRAY_ARRAY_UDINT_AUTO[3][5] := ARRAY_ARRAY_UDINT_AUTO[3][5] + 1;
    ARRAY_ARRAY_UDINT_AUTO[3][6] := ARRAY_ARRAY_UDINT_AUTO[3][6] + 1;
    ARRAY_ARRAY_UDINT_AUTO[3][7] := ARRAY_ARRAY_UDINT_AUTO[3][7] + 1;
    ARRAY_ARRAY_UDINT_AUTO[3][8] := ARRAY_ARRAY_UDINT_AUTO[3][8] + 1;
    ARRAY_ARRAY_UDINT_AUTO[3][9] := ARRAY_ARRAY_UDINT_AUTO[3][9] + 1;

    ARRAY_ARRAY_UDINT_AUTO[4][0] := ARRAY_ARRAY_UDINT_AUTO[4][0] + 1;
    ARRAY_ARRAY_UDINT_AUTO[4][1] := ARRAY_ARRAY_UDINT_AUTO[4][1] + 1;
    ARRAY_ARRAY_UDINT_AUTO[4][2] := ARRAY_ARRAY_UDINT_AUTO[4][2] + 1;
    ARRAY_ARRAY_UDINT_AUTO[4][3] := ARRAY_ARRAY_UDINT_AUTO[4][3] + 1;
    ARRAY_ARRAY_UDINT_AUTO[4][4] := ARRAY_ARRAY_UDINT_AUTO[4][4] + 1;
    ARRAY_ARRAY_UDINT_AUTO[4][5] := ARRAY_ARRAY_UDINT_AUTO[4][5] + 1;
    ARRAY_ARRAY_UDINT_AUTO[4][6] := ARRAY_ARRAY_UDINT_AUTO[4][6] + 1;
    ARRAY_ARRAY_UDINT_AUTO[4][7] := ARRAY_ARRAY_UDINT_AUTO[4][7] + 1;
    ARRAY_ARRAY_UDINT_AUTO[4][8] := ARRAY_ARRAY_UDINT_AUTO[4][8] + 1;
    ARRAY_ARRAY_UDINT_AUTO[4][9] := ARRAY_ARRAY_UDINT_AUTO[4][9] + 1;

    ARRAY_ARRAY_UDINT_AUTO[5][0] := ARRAY_ARRAY_UDINT_AUTO[5][0] + 1;
    ARRAY_ARRAY_UDINT_AUTO[5][1] := ARRAY_ARRAY_UDINT_AUTO[5][1] + 1;
    ARRAY_ARRAY_UDINT_AUTO[5][2] := ARRAY_ARRAY_UDINT_AUTO[5][2] + 1;
    ARRAY_ARRAY_UDINT_AUTO[5][3] := ARRAY_ARRAY_UDINT_AUTO[5][3] + 1;
    ARRAY_ARRAY_UDINT_AUTO[5][4] := ARRAY_ARRAY_UDINT_AUTO[5][4] + 1;
    ARRAY_ARRAY_UDINT_AUTO[5][5] := ARRAY_ARRAY_UDINT_AUTO[5][5] + 1;
    ARRAY_ARRAY_UDINT_AUTO[5][6] := ARRAY_ARRAY_UDINT_AUTO[5][6] + 1;
    ARRAY_ARRAY_UDINT_AUTO[5][7] := ARRAY_ARRAY_UDINT_AUTO[5][7] + 1;
    ARRAY_ARRAY_UDINT_AUTO[5][8] := ARRAY_ARRAY_UDINT_AUTO[5][8] + 1;
    ARRAY_ARRAY_UDINT_AUTO[5][9] := ARRAY_ARRAY_UDINT_AUTO[5][9] + 1;

    ARRAY_ARRAY_UDINT_AUTO[6][0] := ARRAY_ARRAY_UDINT_AUTO[6][0] + 1;
    ARRAY_ARRAY_UDINT_AUTO[6][1] := ARRAY_ARRAY_UDINT_AUTO[6][1] + 1;
    ARRAY_ARRAY_UDINT_AUTO[6][2] := ARRAY_ARRAY_UDINT_AUTO[6][2] + 1;
    ARRAY_ARRAY_UDINT_AUTO[6][3] := ARRAY_ARRAY_UDINT_AUTO[6][3] + 1;
    ARRAY_ARRAY_UDINT_AUTO[6][4] := ARRAY_ARRAY_UDINT_AUTO[6][4] + 1;
    ARRAY_ARRAY_UDINT_AUTO[6][5] := ARRAY_ARRAY_UDINT_AUTO[6][5] + 1;
    ARRAY_ARRAY_UDINT_AUTO[6][6] := ARRAY_ARRAY_UDINT_AUTO[6][6] + 1;
    ARRAY_ARRAY_UDINT_AUTO[6][7] := ARRAY_ARRAY_UDINT_AUTO[6][7] + 1;
    ARRAY_ARRAY_UDINT_AUTO[6][8] := ARRAY_ARRAY_UDINT_AUTO[6][8] + 1;
    ARRAY_ARRAY_UDINT_AUTO[6][9] := ARRAY_ARRAY_UDINT_AUTO[6][9] + 1;

    ARRAY_ARRAY_UDINT_AUTO[7][0] := ARRAY_ARRAY_UDINT_AUTO[6][0];
    ARRAY_ARRAY_UDINT_AUTO[7][1] := ARRAY_ARRAY_UDINT_AUTO[6][1];
    ARRAY_ARRAY_UDINT_AUTO[7][2] := ARRAY_ARRAY_UDINT_AUTO[6][2];
    ARRAY_ARRAY_UDINT_AUTO[7][3] := ARRAY_ARRAY_UDINT_AUTO[6][3];
    ARRAY_ARRAY_UDINT_AUTO[7][4] := ARRAY_ARRAY_UDINT_AUTO[6][4];
    ARRAY_ARRAY_UDINT_AUTO[7][5] := ARRAY_ARRAY_UDINT_AUTO[6][5];
    ARRAY_ARRAY_UDINT_AUTO[7][6] := ARRAY_ARRAY_UDINT_AUTO[6][6];
    ARRAY_ARRAY_UDINT_AUTO[7][7] := ARRAY_ARRAY_UDINT_AUTO[6][7];
    ARRAY_ARRAY_UDINT_AUTO[7][8] := ARRAY_ARRAY_UDINT_AUTO[6][8];
    ARRAY_ARRAY_UDINT_AUTO[7][9] := ARRAY_ARRAY_UDINT_AUTO[6][9];

    ARRAY_ARRAY_UINT_AUTO[0][0] := ARRAY_ARRAY_UINT_AUTO[0][0] + 1;
    ARRAY_ARRAY_UINT_AUTO[0][1] := ARRAY_ARRAY_UINT_AUTO[0][1] + 1;
    ARRAY_ARRAY_UINT_AUTO[0][2] := ARRAY_ARRAY_UINT_AUTO[0][2] + 1;
    ARRAY_ARRAY_UINT_AUTO[0][3] := ARRAY_ARRAY_UINT_AUTO[0][3] + 1;
    ARRAY_ARRAY_UINT_AUTO[0][4] := ARRAY_ARRAY_UINT_AUTO[0][4] + 1;
    ARRAY_ARRAY_UINT_AUTO[0][5] := ARRAY_ARRAY_UINT_AUTO[0][5] + 1;
    ARRAY_ARRAY_UINT_AUTO[0][6] := ARRAY_ARRAY_UINT_AUTO[0][6] + 1;
    ARRAY_ARRAY_UINT_AUTO[0][7] := ARRAY_ARRAY_UINT_AUTO[0][7] + 1;
    ARRAY_ARRAY_UINT_AUTO[0][8] := ARRAY_ARRAY_UINT_AUTO[0][6];
    ARRAY_ARRAY_UINT_AUTO[0][9] := ARRAY_ARRAY_UINT_AUTO[0][7];

    ARRAY_ARRAY_UINT_AUTO[1][0] := ARRAY_ARRAY_UINT_AUTO[1][0] + 1;
    ARRAY_ARRAY_UINT_AUTO[1][1] := ARRAY_ARRAY_UINT_AUTO[1][1] + 1;
    ARRAY_ARRAY_UINT_AUTO[1][2] := ARRAY_ARRAY_UINT_AUTO[1][2] + 1;
    ARRAY_ARRAY_UINT_AUTO[1][3] := ARRAY_ARRAY_UINT_AUTO[1][3] + 1;
    ARRAY_ARRAY_UINT_AUTO[1][4] := ARRAY_ARRAY_UINT_AUTO[1][4] + 1;
    ARRAY_ARRAY_UINT_AUTO[1][5] := ARRAY_ARRAY_UINT_AUTO[1][5] + 1;
    ARRAY_ARRAY_UINT_AUTO[1][6] := ARRAY_ARRAY_UINT_AUTO[1][6] + 1;
    ARRAY_ARRAY_UINT_AUTO[1][7] := ARRAY_ARRAY_UINT_AUTO[1][7] + 1;
    ARRAY_ARRAY_UINT_AUTO[1][8] := ARRAY_ARRAY_UINT_AUTO[1][6];
    ARRAY_ARRAY_UINT_AUTO[1][9] := ARRAY_ARRAY_UINT_AUTO[1][7];

    ARRAY_ARRAY_UINT_AUTO[2][0] := ARRAY_ARRAY_UINT_AUTO[2][0] + 1;
    ARRAY_ARRAY_UINT_AUTO[2][1] := ARRAY_ARRAY_UINT_AUTO[2][1] + 1;
    ARRAY_ARRAY_UINT_AUTO[2][2] := ARRAY_ARRAY_UINT_AUTO[2][2] + 1;
    ARRAY_ARRAY_UINT_AUTO[2][3] := ARRAY_ARRAY_UINT_AUTO[2][3] + 1;
    ARRAY_ARRAY_UINT_AUTO[2][4] := ARRAY_ARRAY_UINT_AUTO[2][4] + 1;
    ARRAY_ARRAY_UINT_AUTO[2][5] := ARRAY_ARRAY_UINT_AUTO[2][5] + 1;
    ARRAY_ARRAY_UINT_AUTO[2][6] := ARRAY_ARRAY_UINT_AUTO[2][6] + 1;
    ARRAY_ARRAY_UINT_AUTO[2][7] := ARRAY_ARRAY_UINT_AUTO[2][7] + 1;
    ARRAY_ARRAY_UINT_AUTO[2][8] := ARRAY_ARRAY_UINT_AUTO[2][8] + 1;
    ARRAY_ARRAY_UINT_AUTO[2][9] := ARRAY_ARRAY_UINT_AUTO[2][9] + 1;

    ARRAY_ARRAY_UINT_AUTO[3][0] := ARRAY_ARRAY_UINT_AUTO[3][0] + 1;
    ARRAY_ARRAY_UINT_AUTO[3][1] := ARRAY_ARRAY_UINT_AUTO[3][1] + 1;
    ARRAY_ARRAY_UINT_AUTO[3][2] := ARRAY_ARRAY_UINT_AUTO[3][2] + 1;
    ARRAY_ARRAY_UINT_AUTO[3][3] := ARRAY_ARRAY_UINT_AUTO[3][3] + 1;
    ARRAY_ARRAY_UINT_AUTO[3][4] := ARRAY_ARRAY_UINT_AUTO[3][4] + 1;
    ARRAY_ARRAY_UINT_AUTO[3][5] := ARRAY_ARRAY_UINT_AUTO[3][5] + 1;
    ARRAY_ARRAY_UINT_AUTO[3][6] := ARRAY_ARRAY_UINT_AUTO[3][6] + 1;
    ARRAY_ARRAY_UINT_AUTO[3][7] := ARRAY_ARRAY_UINT_AUTO[3][7] + 1;
    ARRAY_ARRAY_UINT_AUTO[3][8] := ARRAY_ARRAY_UINT_AUTO[3][8] + 1;
    ARRAY_ARRAY_UINT_AUTO[3][9] := ARRAY_ARRAY_UINT_AUTO[3][9] + 1;

    ARRAY_ARRAY_UINT_AUTO[4][0] := ARRAY_ARRAY_UINT_AUTO[4][0] + 1;
    ARRAY_ARRAY_UINT_AUTO[4][1] := ARRAY_ARRAY_UINT_AUTO[4][1] + 1;
    ARRAY_ARRAY_UINT_AUTO[4][2] := ARRAY_ARRAY_UINT_AUTO[4][2] + 1;
    ARRAY_ARRAY_UINT_AUTO[4][3] := ARRAY_ARRAY_UINT_AUTO[4][3] + 1;
    ARRAY_ARRAY_UINT_AUTO[4][4] := ARRAY_ARRAY_UINT_AUTO[4][4] + 1;
    ARRAY_ARRAY_UINT_AUTO[4][5] := ARRAY_ARRAY_UINT_AUTO[4][5] + 1;
    ARRAY_ARRAY_UINT_AUTO[4][6] := ARRAY_ARRAY_UINT_AUTO[4][6] + 1;
    ARRAY_ARRAY_UINT_AUTO[4][7] := ARRAY_ARRAY_UINT_AUTO[4][7] + 1;
    ARRAY_ARRAY_UINT_AUTO[4][8] := ARRAY_ARRAY_UINT_AUTO[4][8] + 1;
    ARRAY_ARRAY_UINT_AUTO[4][9] := ARRAY_ARRAY_UINT_AUTO[4][9] + 1;

    ARRAY_ARRAY_UINT_AUTO[5][0] := ARRAY_ARRAY_UINT_AUTO[5][0] + 1;
    ARRAY_ARRAY_UINT_AUTO[5][1] := ARRAY_ARRAY_UINT_AUTO[5][1] + 1;
    ARRAY_ARRAY_UINT_AUTO[5][2] := ARRAY_ARRAY_UINT_AUTO[5][2] + 1;
    ARRAY_ARRAY_UINT_AUTO[5][3] := ARRAY_ARRAY_UINT_AUTO[5][3] + 1;
    ARRAY_ARRAY_UINT_AUTO[5][4] := ARRAY_ARRAY_UINT_AUTO[5][4] + 1;
    ARRAY_ARRAY_UINT_AUTO[5][5] := ARRAY_ARRAY_UINT_AUTO[5][5] + 1;
    ARRAY_ARRAY_UINT_AUTO[5][6] := ARRAY_ARRAY_UINT_AUTO[5][6] + 1;
    ARRAY_ARRAY_UINT_AUTO[5][7] := ARRAY_ARRAY_UINT_AUTO[5][7] + 1;
    ARRAY_ARRAY_UINT_AUTO[5][8] := ARRAY_ARRAY_UINT_AUTO[5][8] + 1;
    ARRAY_ARRAY_UINT_AUTO[5][9] := ARRAY_ARRAY_UINT_AUTO[5][9] + 1;

    ARRAY_ARRAY_UINT_AUTO[6][0] := ARRAY_ARRAY_UINT_AUTO[6][0] + 1;
    ARRAY_ARRAY_UINT_AUTO[6][1] := ARRAY_ARRAY_UINT_AUTO[6][1] + 1;
    ARRAY_ARRAY_UINT_AUTO[6][2] := ARRAY_ARRAY_UINT_AUTO[6][2] + 1;
    ARRAY_ARRAY_UINT_AUTO[6][3] := ARRAY_ARRAY_UINT_AUTO[6][3] + 1;
    ARRAY_ARRAY_UINT_AUTO[6][4] := ARRAY_ARRAY_UINT_AUTO[6][4] + 1;
    ARRAY_ARRAY_UINT_AUTO[6][5] := ARRAY_ARRAY_UINT_AUTO[6][5] + 1;
    ARRAY_ARRAY_UINT_AUTO[6][6] := ARRAY_ARRAY_UINT_AUTO[6][6] + 1;
    ARRAY_ARRAY_UINT_AUTO[6][7] := ARRAY_ARRAY_UINT_AUTO[6][7] + 1;
    ARRAY_ARRAY_UINT_AUTO[6][8] := ARRAY_ARRAY_UINT_AUTO[6][8] + 1;
    ARRAY_ARRAY_UINT_AUTO[6][9] := ARRAY_ARRAY_UINT_AUTO[6][9] + 1;

    ARRAY_ARRAY_UINT_AUTO[7][0] := ARRAY_ARRAY_UINT_AUTO[6][0];
    ARRAY_ARRAY_UINT_AUTO[7][1] := ARRAY_ARRAY_UINT_AUTO[6][1];
    ARRAY_ARRAY_UINT_AUTO[7][2] := ARRAY_ARRAY_UINT_AUTO[6][2];
    ARRAY_ARRAY_UINT_AUTO[7][3] := ARRAY_ARRAY_UINT_AUTO[6][3];
    ARRAY_ARRAY_UINT_AUTO[7][4] := ARRAY_ARRAY_UINT_AUTO[6][4];
    ARRAY_ARRAY_UINT_AUTO[7][5] := ARRAY_ARRAY_UINT_AUTO[6][5];
    ARRAY_ARRAY_UINT_AUTO[7][6] := ARRAY_ARRAY_UINT_AUTO[6][6];
    ARRAY_ARRAY_UINT_AUTO[7][7] := ARRAY_ARRAY_UINT_AUTO[6][7];
    ARRAY_ARRAY_UINT_AUTO[7][8] := ARRAY_ARRAY_UINT_AUTO[6][8];
    ARRAY_ARRAY_UINT_AUTO[7][9] := ARRAY_ARRAY_UINT_AUTO[6][9];

    ARRAY_ARRAY_ULINT_AUTO[0][0] := ARRAY_ARRAY_ULINT_AUTO[0][0] + 1;
    ARRAY_ARRAY_ULINT_AUTO[0][1] := ARRAY_ARRAY_ULINT_AUTO[0][1] + 1;
    ARRAY_ARRAY_ULINT_AUTO[0][2] := ARRAY_ARRAY_ULINT_AUTO[0][2] + 1;
    ARRAY_ARRAY_ULINT_AUTO[0][3] := ARRAY_ARRAY_ULINT_AUTO[0][3] + 1;
    ARRAY_ARRAY_ULINT_AUTO[0][4] := ARRAY_ARRAY_ULINT_AUTO[0][4] + 1;
    ARRAY_ARRAY_ULINT_AUTO[0][5] := ARRAY_ARRAY_ULINT_AUTO[0][5] + 1;
    ARRAY_ARRAY_ULINT_AUTO[0][6] := ARRAY_ARRAY_ULINT_AUTO[0][6] + 1;
    ARRAY_ARRAY_ULINT_AUTO[0][7] := ARRAY_ARRAY_ULINT_AUTO[0][7] + 1;
    ARRAY_ARRAY_ULINT_AUTO[0][8] := ARRAY_ARRAY_ULINT_AUTO[0][6];
    ARRAY_ARRAY_ULINT_AUTO[0][9] := ARRAY_ARRAY_ULINT_AUTO[0][7];

    ARRAY_ARRAY_ULINT_AUTO[1][0] := ARRAY_ARRAY_ULINT_AUTO[1][0] + 1;
    ARRAY_ARRAY_ULINT_AUTO[1][1] := ARRAY_ARRAY_ULINT_AUTO[1][1] + 1;
    ARRAY_ARRAY_ULINT_AUTO[1][2] := ARRAY_ARRAY_ULINT_AUTO[1][2] + 1;
    ARRAY_ARRAY_ULINT_AUTO[1][3] := ARRAY_ARRAY_ULINT_AUTO[1][3] + 1;
    ARRAY_ARRAY_ULINT_AUTO[1][4] := ARRAY_ARRAY_ULINT_AUTO[1][4] + 1;
    ARRAY_ARRAY_ULINT_AUTO[1][5] := ARRAY_ARRAY_ULINT_AUTO[1][5] + 1;
    ARRAY_ARRAY_ULINT_AUTO[1][6] := ARRAY_ARRAY_ULINT_AUTO[1][6] + 1;
    ARRAY_ARRAY_ULINT_AUTO[1][7] := ARRAY_ARRAY_ULINT_AUTO[1][7] + 1;
    ARRAY_ARRAY_ULINT_AUTO[1][8] := ARRAY_ARRAY_ULINT_AUTO[1][6];
    ARRAY_ARRAY_ULINT_AUTO[1][9] := ARRAY_ARRAY_ULINT_AUTO[1][7];

    ARRAY_ARRAY_ULINT_AUTO[2][0] := ARRAY_ARRAY_ULINT_AUTO[2][0] + 1;
    ARRAY_ARRAY_ULINT_AUTO[2][1] := ARRAY_ARRAY_ULINT_AUTO[2][1] + 1;
    ARRAY_ARRAY_ULINT_AUTO[2][2] := ARRAY_ARRAY_ULINT_AUTO[2][2] + 1;
    ARRAY_ARRAY_ULINT_AUTO[2][3] := ARRAY_ARRAY_ULINT_AUTO[2][3] + 1;
    ARRAY_ARRAY_ULINT_AUTO[2][4] := ARRAY_ARRAY_ULINT_AUTO[2][4] + 1;
    ARRAY_ARRAY_ULINT_AUTO[2][5] := ARRAY_ARRAY_ULINT_AUTO[2][5] + 1;
    ARRAY_ARRAY_ULINT_AUTO[2][6] := ARRAY_ARRAY_ULINT_AUTO[2][6] + 1;
    ARRAY_ARRAY_ULINT_AUTO[2][7] := ARRAY_ARRAY_ULINT_AUTO[2][7] + 1;
    ARRAY_ARRAY_ULINT_AUTO[2][8] := ARRAY_ARRAY_ULINT_AUTO[2][8] + 1;
    ARRAY_ARRAY_ULINT_AUTO[2][9] := ARRAY_ARRAY_ULINT_AUTO[2][9] + 1;

    ARRAY_ARRAY_ULINT_AUTO[3][0] := ARRAY_ARRAY_ULINT_AUTO[3][0] + 1;
    ARRAY_ARRAY_ULINT_AUTO[3][1] := ARRAY_ARRAY_ULINT_AUTO[3][1] + 1;
    ARRAY_ARRAY_ULINT_AUTO[3][2] := ARRAY_ARRAY_ULINT_AUTO[3][2] + 1;
    ARRAY_ARRAY_ULINT_AUTO[3][3] := ARRAY_ARRAY_ULINT_AUTO[3][3] + 1;
    ARRAY_ARRAY_ULINT_AUTO[3][4] := ARRAY_ARRAY_ULINT_AUTO[3][4] + 1;
    ARRAY_ARRAY_ULINT_AUTO[3][5] := ARRAY_ARRAY_ULINT_AUTO[3][5] + 1;
    ARRAY_ARRAY_ULINT_AUTO[3][6] := ARRAY_ARRAY_ULINT_AUTO[3][6] + 1;
    ARRAY_ARRAY_ULINT_AUTO[3][7] := ARRAY_ARRAY_ULINT_AUTO[3][7] + 1;
    ARRAY_ARRAY_ULINT_AUTO[3][8] := ARRAY_ARRAY_ULINT_AUTO[3][8] + 1;
    ARRAY_ARRAY_ULINT_AUTO[3][9] := ARRAY_ARRAY_ULINT_AUTO[3][8] + 1;

    ARRAY_ARRAY_ULINT_AUTO[4][0] := ARRAY_ARRAY_ULINT_AUTO[4][0] + 1;
    ARRAY_ARRAY_ULINT_AUTO[4][1] := ARRAY_ARRAY_ULINT_AUTO[4][1] + 1;
    ARRAY_ARRAY_ULINT_AUTO[4][2] := ARRAY_ARRAY_ULINT_AUTO[4][2] + 1;
    ARRAY_ARRAY_ULINT_AUTO[4][3] := ARRAY_ARRAY_ULINT_AUTO[4][3] + 1;
    ARRAY_ARRAY_ULINT_AUTO[4][4] := ARRAY_ARRAY_ULINT_AUTO[4][4] + 1;
    ARRAY_ARRAY_ULINT_AUTO[4][5] := ARRAY_ARRAY_ULINT_AUTO[4][5] + 1;
    ARRAY_ARRAY_ULINT_AUTO[4][6] := ARRAY_ARRAY_ULINT_AUTO[4][6] + 1;
    ARRAY_ARRAY_ULINT_AUTO[4][7] := ARRAY_ARRAY_ULINT_AUTO[4][7] + 1;
    ARRAY_ARRAY_ULINT_AUTO[4][8] := ARRAY_ARRAY_ULINT_AUTO[4][8] + 1;
    ARRAY_ARRAY_ULINT_AUTO[4][9] := ARRAY_ARRAY_ULINT_AUTO[4][9] + 1;

    ARRAY_ARRAY_ULINT_AUTO[5][0] := ARRAY_ARRAY_ULINT_AUTO[5][0] + 1;
    ARRAY_ARRAY_ULINT_AUTO[5][1] := ARRAY_ARRAY_ULINT_AUTO[5][1] + 1;
    ARRAY_ARRAY_ULINT_AUTO[5][2] := ARRAY_ARRAY_ULINT_AUTO[5][2] + 1;
    ARRAY_ARRAY_ULINT_AUTO[5][3] := ARRAY_ARRAY_ULINT_AUTO[5][3] + 1;
    ARRAY_ARRAY_ULINT_AUTO[5][4] := ARRAY_ARRAY_ULINT_AUTO[5][4] + 1;
    ARRAY_ARRAY_ULINT_AUTO[5][5] := ARRAY_ARRAY_ULINT_AUTO[5][5] + 1;
    ARRAY_ARRAY_ULINT_AUTO[5][6] := ARRAY_ARRAY_ULINT_AUTO[5][6] + 1;
    ARRAY_ARRAY_ULINT_AUTO[5][7] := ARRAY_ARRAY_ULINT_AUTO[5][7] + 1;
    ARRAY_ARRAY_ULINT_AUTO[5][8] := ARRAY_ARRAY_ULINT_AUTO[5][8] + 1;
    ARRAY_ARRAY_ULINT_AUTO[5][9] := ARRAY_ARRAY_ULINT_AUTO[5][9] + 1;

    ARRAY_ARRAY_ULINT_AUTO[6][0] := ARRAY_ARRAY_ULINT_AUTO[6][0] + 1;
    ARRAY_ARRAY_ULINT_AUTO[6][1] := ARRAY_ARRAY_ULINT_AUTO[6][1] + 1;
    ARRAY_ARRAY_ULINT_AUTO[6][2] := ARRAY_ARRAY_ULINT_AUTO[6][2] + 1;
    ARRAY_ARRAY_ULINT_AUTO[6][3] := ARRAY_ARRAY_ULINT_AUTO[6][3] + 1;
    ARRAY_ARRAY_ULINT_AUTO[6][4] := ARRAY_ARRAY_ULINT_AUTO[6][4] + 1;
    ARRAY_ARRAY_ULINT_AUTO[6][5] := ARRAY_ARRAY_ULINT_AUTO[6][5] + 1;
    ARRAY_ARRAY_ULINT_AUTO[6][6] := ARRAY_ARRAY_ULINT_AUTO[6][6] + 1;
    ARRAY_ARRAY_ULINT_AUTO[6][7] := ARRAY_ARRAY_ULINT_AUTO[6][7] + 1;
    ARRAY_ARRAY_ULINT_AUTO[6][8] := ARRAY_ARRAY_ULINT_AUTO[6][8] + 1;
    ARRAY_ARRAY_ULINT_AUTO[6][9] := ARRAY_ARRAY_ULINT_AUTO[6][9] + 1;

    ARRAY_ARRAY_ULINT_AUTO[7][0] := ARRAY_ARRAY_ULINT_AUTO[6][0];
    ARRAY_ARRAY_ULINT_AUTO[7][1] := ARRAY_ARRAY_ULINT_AUTO[6][1];
    ARRAY_ARRAY_ULINT_AUTO[7][2] := ARRAY_ARRAY_ULINT_AUTO[6][2];
    ARRAY_ARRAY_ULINT_AUTO[7][3] := ARRAY_ARRAY_ULINT_AUTO[6][3];
    ARRAY_ARRAY_ULINT_AUTO[7][4] := ARRAY_ARRAY_ULINT_AUTO[6][4];
    ARRAY_ARRAY_ULINT_AUTO[7][5] := ARRAY_ARRAY_ULINT_AUTO[6][5];
    ARRAY_ARRAY_ULINT_AUTO[7][6] := ARRAY_ARRAY_ULINT_AUTO[6][6];
    ARRAY_ARRAY_ULINT_AUTO[7][7] := ARRAY_ARRAY_ULINT_AUTO[6][7];
    ARRAY_ARRAY_ULINT_AUTO[7][8] := ARRAY_ARRAY_ULINT_AUTO[6][8];
    ARRAY_ARRAY_ULINT_AUTO[7][9] := ARRAY_ARRAY_ULINT_AUTO[6][9];

    ARRAY_ARRAY_USINT_AUTO[0][0] := ARRAY_ARRAY_USINT_AUTO[0][0] + 1;
    ARRAY_ARRAY_USINT_AUTO[0][1] := ARRAY_ARRAY_USINT_AUTO[0][1] + 1;
    ARRAY_ARRAY_USINT_AUTO[0][2] := ARRAY_ARRAY_USINT_AUTO[0][2] + 1;
    ARRAY_ARRAY_USINT_AUTO[0][3] := ARRAY_ARRAY_USINT_AUTO[0][3] + 1;
    ARRAY_ARRAY_USINT_AUTO[0][4] := ARRAY_ARRAY_USINT_AUTO[0][4] + 1;
    ARRAY_ARRAY_USINT_AUTO[0][5] := ARRAY_ARRAY_USINT_AUTO[0][5] + 1;
    ARRAY_ARRAY_USINT_AUTO[0][6] := ARRAY_ARRAY_USINT_AUTO[0][6] + 1;
    ARRAY_ARRAY_USINT_AUTO[0][7] := ARRAY_ARRAY_USINT_AUTO[0][7] + 1;
    ARRAY_ARRAY_USINT_AUTO[0][8] := ARRAY_ARRAY_USINT_AUTO[0][6];
    ARRAY_ARRAY_USINT_AUTO[0][9] := ARRAY_ARRAY_USINT_AUTO[0][7];

    ARRAY_ARRAY_USINT_AUTO[1][0] := ARRAY_ARRAY_USINT_AUTO[1][0] + 1;
    ARRAY_ARRAY_USINT_AUTO[1][1] := ARRAY_ARRAY_USINT_AUTO[1][1] + 1;
    ARRAY_ARRAY_USINT_AUTO[1][2] := ARRAY_ARRAY_USINT_AUTO[1][2] + 1;
    ARRAY_ARRAY_USINT_AUTO[1][3] := ARRAY_ARRAY_USINT_AUTO[1][3] + 1;
    ARRAY_ARRAY_USINT_AUTO[1][4] := ARRAY_ARRAY_USINT_AUTO[1][4] + 1;
    ARRAY_ARRAY_USINT_AUTO[1][5] := ARRAY_ARRAY_USINT_AUTO[1][5] + 1;
    ARRAY_ARRAY_USINT_AUTO[1][6] := ARRAY_ARRAY_USINT_AUTO[1][6] + 1;
    ARRAY_ARRAY_USINT_AUTO[1][7] := ARRAY_ARRAY_USINT_AUTO[1][7] + 1;
    ARRAY_ARRAY_USINT_AUTO[1][8] := ARRAY_ARRAY_USINT_AUTO[1][6];
    ARRAY_ARRAY_USINT_AUTO[1][9] := ARRAY_ARRAY_USINT_AUTO[1][7];

    ARRAY_ARRAY_USINT_AUTO[2][0] := ARRAY_ARRAY_USINT_AUTO[2][0] + 1;
    ARRAY_ARRAY_USINT_AUTO[2][1] := ARRAY_ARRAY_USINT_AUTO[2][1] + 1;
    ARRAY_ARRAY_USINT_AUTO[2][2] := ARRAY_ARRAY_USINT_AUTO[2][2] + 1;
    ARRAY_ARRAY_USINT_AUTO[2][3] := ARRAY_ARRAY_USINT_AUTO[2][3] + 1;
    ARRAY_ARRAY_USINT_AUTO[2][4] := ARRAY_ARRAY_USINT_AUTO[2][4] + 1;
    ARRAY_ARRAY_USINT_AUTO[2][5] := ARRAY_ARRAY_USINT_AUTO[2][5] + 1;
    ARRAY_ARRAY_USINT_AUTO[2][6] := ARRAY_ARRAY_USINT_AUTO[2][6] + 1;
    ARRAY_ARRAY_USINT_AUTO[2][7] := ARRAY_ARRAY_USINT_AUTO[2][7] + 1;
    ARRAY_ARRAY_USINT_AUTO[2][8] := ARRAY_ARRAY_USINT_AUTO[2][8] + 1;
    ARRAY_ARRAY_USINT_AUTO[2][9] := ARRAY_ARRAY_USINT_AUTO[2][9] + 1;

    ARRAY_ARRAY_USINT_AUTO[3][0] := ARRAY_ARRAY_USINT_AUTO[3][0] + 1;
    ARRAY_ARRAY_USINT_AUTO[3][1] := ARRAY_ARRAY_USINT_AUTO[3][1] + 1;
    ARRAY_ARRAY_USINT_AUTO[3][2] := ARRAY_ARRAY_USINT_AUTO[3][2] + 1;
    ARRAY_ARRAY_USINT_AUTO[3][3] := ARRAY_ARRAY_USINT_AUTO[3][3] + 1;
    ARRAY_ARRAY_USINT_AUTO[3][4] := ARRAY_ARRAY_USINT_AUTO[3][4] + 1;
    ARRAY_ARRAY_USINT_AUTO[3][5] := ARRAY_ARRAY_USINT_AUTO[3][5] + 1;
    ARRAY_ARRAY_USINT_AUTO[3][6] := ARRAY_ARRAY_USINT_AUTO[3][6] + 1;
    ARRAY_ARRAY_USINT_AUTO[3][7] := ARRAY_ARRAY_USINT_AUTO[3][7] + 1;
    ARRAY_ARRAY_USINT_AUTO[3][8] := ARRAY_ARRAY_USINT_AUTO[3][8] + 1;
    ARRAY_ARRAY_USINT_AUTO[3][9] := ARRAY_ARRAY_USINT_AUTO[3][8] + 1;

    ARRAY_ARRAY_USINT_AUTO[4][0] := ARRAY_ARRAY_USINT_AUTO[4][0] + 1;
    ARRAY_ARRAY_USINT_AUTO[4][1] := ARRAY_ARRAY_USINT_AUTO[4][1] + 1;
    ARRAY_ARRAY_USINT_AUTO[4][2] := ARRAY_ARRAY_USINT_AUTO[4][2] + 1;
    ARRAY_ARRAY_USINT_AUTO[4][3] := ARRAY_ARRAY_USINT_AUTO[4][3] + 1;
    ARRAY_ARRAY_USINT_AUTO[4][4] := ARRAY_ARRAY_USINT_AUTO[4][4] + 1;
    ARRAY_ARRAY_USINT_AUTO[4][5] := ARRAY_ARRAY_USINT_AUTO[4][5] + 1;
    ARRAY_ARRAY_USINT_AUTO[4][6] := ARRAY_ARRAY_USINT_AUTO[4][6] + 1;
    ARRAY_ARRAY_USINT_AUTO[4][7] := ARRAY_ARRAY_USINT_AUTO[4][7] + 1;
    ARRAY_ARRAY_USINT_AUTO[4][8] := ARRAY_ARRAY_USINT_AUTO[4][8] + 1;
    ARRAY_ARRAY_USINT_AUTO[4][9] := ARRAY_ARRAY_USINT_AUTO[4][9] + 1;

    ARRAY_ARRAY_USINT_AUTO[5][0] := ARRAY_ARRAY_USINT_AUTO[5][0] + 1;
    ARRAY_ARRAY_USINT_AUTO[5][1] := ARRAY_ARRAY_USINT_AUTO[5][1] + 1;
    ARRAY_ARRAY_USINT_AUTO[5][2] := ARRAY_ARRAY_USINT_AUTO[5][2] + 1;
    ARRAY_ARRAY_USINT_AUTO[5][3] := ARRAY_ARRAY_USINT_AUTO[5][3] + 1;
    ARRAY_ARRAY_USINT_AUTO[5][4] := ARRAY_ARRAY_USINT_AUTO[5][4] + 1;
    ARRAY_ARRAY_USINT_AUTO[5][5] := ARRAY_ARRAY_USINT_AUTO[5][5] + 1;
    ARRAY_ARRAY_USINT_AUTO[5][6] := ARRAY_ARRAY_USINT_AUTO[5][6] + 1;
    ARRAY_ARRAY_USINT_AUTO[5][7] := ARRAY_ARRAY_USINT_AUTO[5][7] + 1;
    ARRAY_ARRAY_USINT_AUTO[5][8] := ARRAY_ARRAY_USINT_AUTO[5][8] + 1;
    ARRAY_ARRAY_USINT_AUTO[5][9] := ARRAY_ARRAY_USINT_AUTO[5][9] + 1;

    ARRAY_ARRAY_USINT_AUTO[6][0] := ARRAY_ARRAY_USINT_AUTO[6][0] + 1;
    ARRAY_ARRAY_USINT_AUTO[6][1] := ARRAY_ARRAY_USINT_AUTO[6][1] + 1;
    ARRAY_ARRAY_USINT_AUTO[6][2] := ARRAY_ARRAY_USINT_AUTO[6][2] + 1;
    ARRAY_ARRAY_USINT_AUTO[6][3] := ARRAY_ARRAY_USINT_AUTO[6][3] + 1;
    ARRAY_ARRAY_USINT_AUTO[6][4] := ARRAY_ARRAY_USINT_AUTO[6][4] + 1;
    ARRAY_ARRAY_USINT_AUTO[6][5] := ARRAY_ARRAY_USINT_AUTO[6][5] + 1;
    ARRAY_ARRAY_USINT_AUTO[6][6] := ARRAY_ARRAY_USINT_AUTO[6][6] + 1;
    ARRAY_ARRAY_USINT_AUTO[6][7] := ARRAY_ARRAY_USINT_AUTO[6][7] + 1;
    ARRAY_ARRAY_USINT_AUTO[6][8] := ARRAY_ARRAY_USINT_AUTO[6][8] + 1;
    ARRAY_ARRAY_USINT_AUTO[6][9] := ARRAY_ARRAY_USINT_AUTO[6][9] + 1;

    ARRAY_ARRAY_USINT_AUTO[7][0] := ARRAY_ARRAY_USINT_AUTO[6][0];
    ARRAY_ARRAY_USINT_AUTO[7][1] := ARRAY_ARRAY_USINT_AUTO[6][1];
    ARRAY_ARRAY_USINT_AUTO[7][2] := ARRAY_ARRAY_USINT_AUTO[6][2];
    ARRAY_ARRAY_USINT_AUTO[7][3] := ARRAY_ARRAY_USINT_AUTO[6][3];
    ARRAY_ARRAY_USINT_AUTO[7][4] := ARRAY_ARRAY_USINT_AUTO[6][4];
    ARRAY_ARRAY_USINT_AUTO[7][5] := ARRAY_ARRAY_USINT_AUTO[6][5];
    ARRAY_ARRAY_USINT_AUTO[7][6] := ARRAY_ARRAY_USINT_AUTO[6][6];
    ARRAY_ARRAY_USINT_AUTO[7][7] := ARRAY_ARRAY_USINT_AUTO[6][7];
    ARRAY_ARRAY_USINT_AUTO[7][8] := ARRAY_ARRAY_USINT_AUTO[6][8];
    ARRAY_ARRAY_USINT_AUTO[7][9] := ARRAY_ARRAY_USINT_AUTO[6][9];

    ARRAY_ARRAY_WORD_AUTO[0][0] := ARRAY_ARRAY_WORD_AUTO[0][0] + 1;
    ARRAY_ARRAY_WORD_AUTO[0][1] := ARRAY_ARRAY_WORD_AUTO[0][1] + 1;
    ARRAY_ARRAY_WORD_AUTO[0][2] := ARRAY_ARRAY_WORD_AUTO[0][2] + 1;
    ARRAY_ARRAY_WORD_AUTO[0][3] := ARRAY_ARRAY_WORD_AUTO[0][3] + 1;
    ARRAY_ARRAY_WORD_AUTO[0][4] := ARRAY_ARRAY_WORD_AUTO[0][4] + 1;
    ARRAY_ARRAY_WORD_AUTO[0][5] := ARRAY_ARRAY_WORD_AUTO[0][5] + 1;
    ARRAY_ARRAY_WORD_AUTO[0][6] := ARRAY_ARRAY_WORD_AUTO[0][6] + 1;
    ARRAY_ARRAY_WORD_AUTO[0][7] := ARRAY_ARRAY_WORD_AUTO[0][7] + 1;
    ARRAY_ARRAY_WORD_AUTO[0][8] := ARRAY_ARRAY_WORD_AUTO[0][6];
    ARRAY_ARRAY_WORD_AUTO[0][9] := ARRAY_ARRAY_WORD_AUTO[0][7];

    ARRAY_ARRAY_WORD_AUTO[1][0] := ARRAY_ARRAY_WORD_AUTO[1][0] + 1;
    ARRAY_ARRAY_WORD_AUTO[1][1] := ARRAY_ARRAY_WORD_AUTO[1][1] + 1;
    ARRAY_ARRAY_WORD_AUTO[1][2] := ARRAY_ARRAY_WORD_AUTO[1][2] + 1;
    ARRAY_ARRAY_WORD_AUTO[1][3] := ARRAY_ARRAY_WORD_AUTO[1][3] + 1;
    ARRAY_ARRAY_WORD_AUTO[1][4] := ARRAY_ARRAY_WORD_AUTO[1][4] + 1;
    ARRAY_ARRAY_WORD_AUTO[1][5] := ARRAY_ARRAY_WORD_AUTO[1][5] + 1;
    ARRAY_ARRAY_WORD_AUTO[1][6] := ARRAY_ARRAY_WORD_AUTO[1][6] + 1;
    ARRAY_ARRAY_WORD_AUTO[1][7] := ARRAY_ARRAY_WORD_AUTO[1][7] + 1;
    ARRAY_ARRAY_WORD_AUTO[1][8] := ARRAY_ARRAY_WORD_AUTO[1][6];
    ARRAY_ARRAY_WORD_AUTO[1][9] := ARRAY_ARRAY_WORD_AUTO[1][7];

    ARRAY_ARRAY_WORD_AUTO[2][0] := ARRAY_ARRAY_WORD_AUTO[2][0] + 1;
    ARRAY_ARRAY_WORD_AUTO[2][1] := ARRAY_ARRAY_WORD_AUTO[2][1] + 1;
    ARRAY_ARRAY_WORD_AUTO[2][2] := ARRAY_ARRAY_WORD_AUTO[2][2] + 1;
    ARRAY_ARRAY_WORD_AUTO[2][3] := ARRAY_ARRAY_WORD_AUTO[2][3] + 1;
    ARRAY_ARRAY_WORD_AUTO[2][4] := ARRAY_ARRAY_WORD_AUTO[2][4] + 1;
    ARRAY_ARRAY_WORD_AUTO[2][5] := ARRAY_ARRAY_WORD_AUTO[2][5] + 1;
    ARRAY_ARRAY_WORD_AUTO[2][6] := ARRAY_ARRAY_WORD_AUTO[2][6] + 1;
    ARRAY_ARRAY_WORD_AUTO[2][7] := ARRAY_ARRAY_WORD_AUTO[2][7] + 1;
    ARRAY_ARRAY_WORD_AUTO[2][8] := ARRAY_ARRAY_WORD_AUTO[2][8] + 1;
    ARRAY_ARRAY_WORD_AUTO[2][9] := ARRAY_ARRAY_WORD_AUTO[2][9] + 1;

    ARRAY_ARRAY_WORD_AUTO[3][0] := ARRAY_ARRAY_WORD_AUTO[3][0] + 1;
    ARRAY_ARRAY_WORD_AUTO[3][1] := ARRAY_ARRAY_WORD_AUTO[3][1] + 1;
    ARRAY_ARRAY_WORD_AUTO[3][2] := ARRAY_ARRAY_WORD_AUTO[3][2] + 1;
    ARRAY_ARRAY_WORD_AUTO[3][3] := ARRAY_ARRAY_WORD_AUTO[3][3] + 1;
    ARRAY_ARRAY_WORD_AUTO[3][4] := ARRAY_ARRAY_WORD_AUTO[3][4] + 1;
    ARRAY_ARRAY_WORD_AUTO[3][5] := ARRAY_ARRAY_WORD_AUTO[3][5] + 1;
    ARRAY_ARRAY_WORD_AUTO[3][6] := ARRAY_ARRAY_WORD_AUTO[3][6] + 1;
    ARRAY_ARRAY_WORD_AUTO[3][7] := ARRAY_ARRAY_WORD_AUTO[3][7] + 1;
    ARRAY_ARRAY_WORD_AUTO[3][8] := ARRAY_ARRAY_WORD_AUTO[3][8] + 1;
    ARRAY_ARRAY_WORD_AUTO[3][9] := ARRAY_ARRAY_WORD_AUTO[3][9] + 1;

    ARRAY_ARRAY_WORD_AUTO[4][0] := ARRAY_ARRAY_WORD_AUTO[4][0] + 1;
    ARRAY_ARRAY_WORD_AUTO[4][1] := ARRAY_ARRAY_WORD_AUTO[4][1] + 1;
    ARRAY_ARRAY_WORD_AUTO[4][2] := ARRAY_ARRAY_WORD_AUTO[4][2] + 1;
    ARRAY_ARRAY_WORD_AUTO[4][3] := ARRAY_ARRAY_WORD_AUTO[4][3] + 1;
    ARRAY_ARRAY_WORD_AUTO[4][4] := ARRAY_ARRAY_WORD_AUTO[4][4] + 1;
    ARRAY_ARRAY_WORD_AUTO[4][5] := ARRAY_ARRAY_WORD_AUTO[4][5] + 1;
    ARRAY_ARRAY_WORD_AUTO[4][6] := ARRAY_ARRAY_WORD_AUTO[4][6] + 1;
    ARRAY_ARRAY_WORD_AUTO[4][7] := ARRAY_ARRAY_WORD_AUTO[4][7] + 1;
    ARRAY_ARRAY_WORD_AUTO[4][8] := ARRAY_ARRAY_WORD_AUTO[4][8] + 1;
    ARRAY_ARRAY_WORD_AUTO[4][9] := ARRAY_ARRAY_WORD_AUTO[4][9] + 1;

    ARRAY_ARRAY_WORD_AUTO[5][0] := ARRAY_ARRAY_WORD_AUTO[5][0] + 1;
    ARRAY_ARRAY_WORD_AUTO[5][1] := ARRAY_ARRAY_WORD_AUTO[5][1] + 1;
    ARRAY_ARRAY_WORD_AUTO[5][2] := ARRAY_ARRAY_WORD_AUTO[5][2] + 1;
    ARRAY_ARRAY_WORD_AUTO[5][3] := ARRAY_ARRAY_WORD_AUTO[5][3] + 1;
    ARRAY_ARRAY_WORD_AUTO[5][4] := ARRAY_ARRAY_WORD_AUTO[5][4] + 1;
    ARRAY_ARRAY_WORD_AUTO[5][5] := ARRAY_ARRAY_WORD_AUTO[5][5] + 1;
    ARRAY_ARRAY_WORD_AUTO[5][6] := ARRAY_ARRAY_WORD_AUTO[5][6] + 1;
    ARRAY_ARRAY_WORD_AUTO[5][7] := ARRAY_ARRAY_WORD_AUTO[5][7] + 1;
    ARRAY_ARRAY_WORD_AUTO[5][8] := ARRAY_ARRAY_WORD_AUTO[5][8] + 1;
    ARRAY_ARRAY_WORD_AUTO[5][9] := ARRAY_ARRAY_WORD_AUTO[5][9] + 1;

    ARRAY_ARRAY_WORD_AUTO[6][0] := ARRAY_ARRAY_WORD_AUTO[6][0] + 1;
    ARRAY_ARRAY_WORD_AUTO[6][1] := ARRAY_ARRAY_WORD_AUTO[6][1] + 1;
    ARRAY_ARRAY_WORD_AUTO[6][2] := ARRAY_ARRAY_WORD_AUTO[6][2] + 1;
    ARRAY_ARRAY_WORD_AUTO[6][3] := ARRAY_ARRAY_WORD_AUTO[6][3] + 1;
    ARRAY_ARRAY_WORD_AUTO[6][4] := ARRAY_ARRAY_WORD_AUTO[6][4] + 1;
    ARRAY_ARRAY_WORD_AUTO[6][5] := ARRAY_ARRAY_WORD_AUTO[6][5] + 1;
    ARRAY_ARRAY_WORD_AUTO[6][6] := ARRAY_ARRAY_WORD_AUTO[6][6] + 1;
    ARRAY_ARRAY_WORD_AUTO[6][7] := ARRAY_ARRAY_WORD_AUTO[6][7] + 1;
    ARRAY_ARRAY_WORD_AUTO[6][8] := ARRAY_ARRAY_WORD_AUTO[6][8] + 1;
    ARRAY_ARRAY_WORD_AUTO[6][9] := ARRAY_ARRAY_WORD_AUTO[6][9] + 1;

    ARRAY_ARRAY_WORD_AUTO[7][0] := ARRAY_ARRAY_WORD_AUTO[6][0];
    ARRAY_ARRAY_WORD_AUTO[7][1] := ARRAY_ARRAY_WORD_AUTO[6][1];
    ARRAY_ARRAY_WORD_AUTO[7][2] := ARRAY_ARRAY_WORD_AUTO[6][2];
    ARRAY_ARRAY_WORD_AUTO[7][3] := ARRAY_ARRAY_WORD_AUTO[6][3];
    ARRAY_ARRAY_WORD_AUTO[7][4] := ARRAY_ARRAY_WORD_AUTO[6][4];
    ARRAY_ARRAY_WORD_AUTO[7][5] := ARRAY_ARRAY_WORD_AUTO[6][5];
    ARRAY_ARRAY_WORD_AUTO[7][6] := ARRAY_ARRAY_WORD_AUTO[6][6];
    ARRAY_ARRAY_WORD_AUTO[7][7] := ARRAY_ARRAY_WORD_AUTO[6][7];
    ARRAY_ARRAY_WORD_AUTO[7][8] := ARRAY_ARRAY_WORD_AUTO[6][8];
    ARRAY_ARRAY_WORD_AUTO[7][9] := ARRAY_ARRAY_WORD_AUTO[6][9];

END_IF;

END_PROGRAM

(* ---- ManTestArrayStructure.st ---- *)
PROGRAM ManTestArrayStructure

// МАССИВ СТРУКТУР ПРОСТЫХ ТИПОВ
IF TRIGGER_IMP.Q THEN

    ARRAY_SIMPLE_STRUCTURE_RETAIN[0].BOOL_TYPE := NOT ARRAY_SIMPLE_STRUCTURE_RETAIN[0].BOOL_TYPE;
    ARRAY_SIMPLE_STRUCTURE_RETAIN[0].BYTE_TYPE := ARRAY_SIMPLE_STRUCTURE_RETAIN[0].BYTE_TYPE + 1;
    ARRAY_SIMPLE_STRUCTURE_RETAIN[0].DATE_TYPE := ANY_TO_DATE(1445385600 + ARRAY_SIMPLE_STRUCTURE_RETAIN[0].DINT_TYPE * 86400);
    ARRAY_SIMPLE_STRUCTURE_RETAIN[0].DINT_TYPE := ARRAY_SIMPLE_STRUCTURE_RETAIN[0].DINT_TYPE + 1;
    ARRAY_SIMPLE_STRUCTURE_RETAIN[0].DWORD_TYPE := ARRAY_SIMPLE_STRUCTURE_RETAIN[0].DWORD_TYPE + 1;
    ARRAY_SIMPLE_STRUCTURE_RETAIN[0].INT_TYPE := ARRAY_SIMPLE_STRUCTURE_RETAIN[0].INT_TYPE + 1;
    ARRAY_SIMPLE_STRUCTURE_RETAIN[0].LINT_TYPE := ARRAY_SIMPLE_STRUCTURE_RETAIN[0].LINT_TYPE + 1;
    ARRAY_SIMPLE_STRUCTURE_RETAIN[0].LREAL_TYPE := ARRAY_SIMPLE_STRUCTURE_RETAIN[0].LREAL_TYPE + 1;
    ARRAY_SIMPLE_STRUCTURE_RETAIN[0].LWORD_TYPE := ARRAY_SIMPLE_STRUCTURE_RETAIN[0].LWORD_TYPE + 1;
    ARRAY_SIMPLE_STRUCTURE_RETAIN[0].REAL_TYPE := ARRAY_SIMPLE_STRUCTURE_RETAIN[0].REAL_TYPE + 1;
    ARRAY_SIMPLE_STRUCTURE_RETAIN[0].SINT_TYPE := ARRAY_SIMPLE_STRUCTURE_RETAIN[0].SINT_TYPE + 1;
    ARRAY_SIMPLE_STRUCTURE_RETAIN[0].STRING_TYPE := ANY_TO_STRING(ARRAY_SIMPLE_STRUCTURE_RETAIN[0].DINT_TYPE) + ' ' + ANY_TO_STRING(ARRAY_SIMPLE_STRUCTURE_RETAIN[0].TIME_TYPE);
    ARRAY_SIMPLE_STRUCTURE_RETAIN[0].TIME_TYPE := ARRAY_SIMPLE_STRUCTURE_RETAIN[0].TIME_TYPE + PULSE_TIME;
    ARRAY_SIMPLE_STRUCTURE_RETAIN[0].UDINT_TYPE := ARRAY_SIMPLE_STRUCTURE_RETAIN[0].UDINT_TYPE + 1;
    ARRAY_SIMPLE_STRUCTURE_RETAIN[0].UINT_TYPE := ARRAY_SIMPLE_STRUCTURE_RETAIN[0].UINT_TYPE + 1;
    ARRAY_SIMPLE_STRUCTURE_RETAIN[0].ULINT_TYPE := ARRAY_SIMPLE_STRUCTURE_RETAIN[0].ULINT_TYPE + 1;
    ARRAY_SIMPLE_STRUCTURE_RETAIN[0].USINT_TYPE := ARRAY_SIMPLE_STRUCTURE_RETAIN[0].USINT_TYPE + 1;
    ARRAY_SIMPLE_STRUCTURE_RETAIN[0].WORD_TYPE := ARRAY_SIMPLE_STRUCTURE_RETAIN[0].WORD_TYPE + 1;

    ARRAY_SIMPLE_STRUCTURE_RETAIN[1].BOOL_TYPE := NOT ARRAY_SIMPLE_STRUCTURE_RETAIN[1].BOOL_TYPE;
    ARRAY_SIMPLE_STRUCTURE_RETAIN[1].BYTE_TYPE := ARRAY_SIMPLE_STRUCTURE_RETAIN[1].BYTE_TYPE + 1;
    ARRAY_SIMPLE_STRUCTURE_RETAIN[1].DATE_TYPE := ANY_TO_DATE(1445385600 + ARRAY_SIMPLE_STRUCTURE_RETAIN[1].DINT_TYPE * 86400);
    ARRAY_SIMPLE_STRUCTURE_RETAIN[1].DINT_TYPE := ARRAY_SIMPLE_STRUCTURE_RETAIN[1].DINT_TYPE + 1;
    ARRAY_SIMPLE_STRUCTURE_RETAIN[1].DWORD_TYPE := ARRAY_SIMPLE_STRUCTURE_RETAIN[1].DWORD_TYPE + 1;
    ARRAY_SIMPLE_STRUCTURE_RETAIN[1].INT_TYPE := ARRAY_SIMPLE_STRUCTURE_RETAIN[1].INT_TYPE + 1;
    ARRAY_SIMPLE_STRUCTURE_RETAIN[1].LINT_TYPE := ARRAY_SIMPLE_STRUCTURE_RETAIN[1].LINT_TYPE + 1;
    ARRAY_SIMPLE_STRUCTURE_RETAIN[1].LREAL_TYPE := ARRAY_SIMPLE_STRUCTURE_RETAIN[1].LREAL_TYPE + 1;
    ARRAY_SIMPLE_STRUCTURE_RETAIN[1].LWORD_TYPE := ARRAY_SIMPLE_STRUCTURE_RETAIN[1].LWORD_TYPE + 1;
    ARRAY_SIMPLE_STRUCTURE_RETAIN[1].REAL_TYPE := ARRAY_SIMPLE_STRUCTURE_RETAIN[1].REAL_TYPE + 1;
    ARRAY_SIMPLE_STRUCTURE_RETAIN[1].SINT_TYPE := ARRAY_SIMPLE_STRUCTURE_RETAIN[1].SINT_TYPE + 1;
    ARRAY_SIMPLE_STRUCTURE_RETAIN[1].STRING_TYPE := ANY_TO_STRING(ARRAY_SIMPLE_STRUCTURE_RETAIN[1].DINT_TYPE) + ' ' + ANY_TO_STRING(ARRAY_SIMPLE_STRUCTURE_RETAIN[1].TIME_TYPE);
    ARRAY_SIMPLE_STRUCTURE_RETAIN[1].TIME_TYPE := ARRAY_SIMPLE_STRUCTURE_RETAIN[1].TIME_TYPE + PULSE_TIME;
    ARRAY_SIMPLE_STRUCTURE_RETAIN[1].UDINT_TYPE := ARRAY_SIMPLE_STRUCTURE_RETAIN[1].UDINT_TYPE + 1;
    ARRAY_SIMPLE_STRUCTURE_RETAIN[1].UINT_TYPE := ARRAY_SIMPLE_STRUCTURE_RETAIN[1].UINT_TYPE + 1;
    ARRAY_SIMPLE_STRUCTURE_RETAIN[1].ULINT_TYPE := ARRAY_SIMPLE_STRUCTURE_RETAIN[1].ULINT_TYPE + 1;
    ARRAY_SIMPLE_STRUCTURE_RETAIN[1].USINT_TYPE := ARRAY_SIMPLE_STRUCTURE_RETAIN[1].USINT_TYPE + 1;
    ARRAY_SIMPLE_STRUCTURE_RETAIN[1].WORD_TYPE := ARRAY_SIMPLE_STRUCTURE_RETAIN[1].WORD_TYPE + 1;

    ARRAY_SIMPLE_STRUCTURE_RETAIN[2].BOOL_TYPE := NOT ARRAY_SIMPLE_STRUCTURE_RETAIN[2].BOOL_TYPE;
    ARRAY_SIMPLE_STRUCTURE_RETAIN[2].BYTE_TYPE := ARRAY_SIMPLE_STRUCTURE_RETAIN[2].BYTE_TYPE + 1;
    ARRAY_SIMPLE_STRUCTURE_RETAIN[2].DATE_TYPE := ANY_TO_DATE(1445385600 + ARRAY_SIMPLE_STRUCTURE_RETAIN[2].DINT_TYPE * 86400);
    ARRAY_SIMPLE_STRUCTURE_RETAIN[2].DINT_TYPE := ARRAY_SIMPLE_STRUCTURE_RETAIN[2].DINT_TYPE + 1;
    ARRAY_SIMPLE_STRUCTURE_RETAIN[2].DWORD_TYPE := ARRAY_SIMPLE_STRUCTURE_RETAIN[2].DWORD_TYPE + 1;
    ARRAY_SIMPLE_STRUCTURE_RETAIN[2].INT_TYPE := ARRAY_SIMPLE_STRUCTURE_RETAIN[2].INT_TYPE + 1;
    ARRAY_SIMPLE_STRUCTURE_RETAIN[2].LINT_TYPE := ARRAY_SIMPLE_STRUCTURE_RETAIN[2].LINT_TYPE + 1;
    ARRAY_SIMPLE_STRUCTURE_RETAIN[2].LREAL_TYPE := ARRAY_SIMPLE_STRUCTURE_RETAIN[2].LREAL_TYPE + 1;
    ARRAY_SIMPLE_STRUCTURE_RETAIN[2].LWORD_TYPE := ARRAY_SIMPLE_STRUCTURE_RETAIN[2].LWORD_TYPE + 1;
    ARRAY_SIMPLE_STRUCTURE_RETAIN[2].REAL_TYPE := ARRAY_SIMPLE_STRUCTURE_RETAIN[2].REAL_TYPE + 1;
    ARRAY_SIMPLE_STRUCTURE_RETAIN[2].SINT_TYPE := ARRAY_SIMPLE_STRUCTURE_RETAIN[2].SINT_TYPE + 1;
    ARRAY_SIMPLE_STRUCTURE_RETAIN[2].STRING_TYPE := ANY_TO_STRING(ARRAY_SIMPLE_STRUCTURE_RETAIN[2].DINT_TYPE) + ' ' + ANY_TO_STRING(ARRAY_SIMPLE_STRUCTURE_RETAIN[2].TIME_TYPE);
    ARRAY_SIMPLE_STRUCTURE_RETAIN[2].TIME_TYPE := ARRAY_SIMPLE_STRUCTURE_RETAIN[2].TIME_TYPE + PULSE_TIME;
    ARRAY_SIMPLE_STRUCTURE_RETAIN[2].UDINT_TYPE := ARRAY_SIMPLE_STRUCTURE_RETAIN[2].UDINT_TYPE + 1;
    ARRAY_SIMPLE_STRUCTURE_RETAIN[2].UINT_TYPE := ARRAY_SIMPLE_STRUCTURE_RETAIN[2].UINT_TYPE + 1;
    ARRAY_SIMPLE_STRUCTURE_RETAIN[2].ULINT_TYPE := ARRAY_SIMPLE_STRUCTURE_RETAIN[2].ULINT_TYPE + 1;
    ARRAY_SIMPLE_STRUCTURE_RETAIN[2].USINT_TYPE := ARRAY_SIMPLE_STRUCTURE_RETAIN[2].USINT_TYPE + 1;
    ARRAY_SIMPLE_STRUCTURE_RETAIN[2].WORD_TYPE := ARRAY_SIMPLE_STRUCTURE_RETAIN[2].WORD_TYPE + 1;

    ARRAY_SIMPLE_STRUCTURE_RETAIN[3].BOOL_TYPE := NOT ARRAY_SIMPLE_STRUCTURE_RETAIN[3].BOOL_TYPE;
    ARRAY_SIMPLE_STRUCTURE_RETAIN[3].BYTE_TYPE := ARRAY_SIMPLE_STRUCTURE_RETAIN[3].BYTE_TYPE + 1;
    ARRAY_SIMPLE_STRUCTURE_RETAIN[3].DATE_TYPE := ANY_TO_DATE(1445385600 + ARRAY_SIMPLE_STRUCTURE_RETAIN[3].DINT_TYPE * 86400);
    ARRAY_SIMPLE_STRUCTURE_RETAIN[3].DINT_TYPE := ARRAY_SIMPLE_STRUCTURE_RETAIN[3].DINT_TYPE + 1;
    ARRAY_SIMPLE_STRUCTURE_RETAIN[3].DWORD_TYPE := ARRAY_SIMPLE_STRUCTURE_RETAIN[3].DWORD_TYPE + 1;
    ARRAY_SIMPLE_STRUCTURE_RETAIN[3].INT_TYPE := ARRAY_SIMPLE_STRUCTURE_RETAIN[3].INT_TYPE + 1;
    ARRAY_SIMPLE_STRUCTURE_RETAIN[3].LINT_TYPE := ARRAY_SIMPLE_STRUCTURE_RETAIN[3].LINT_TYPE + 1;
    ARRAY_SIMPLE_STRUCTURE_RETAIN[3].LREAL_TYPE := ARRAY_SIMPLE_STRUCTURE_RETAIN[3].LREAL_TYPE + 1;
    ARRAY_SIMPLE_STRUCTURE_RETAIN[3].LWORD_TYPE := ARRAY_SIMPLE_STRUCTURE_RETAIN[3].LWORD_TYPE + 1;
    ARRAY_SIMPLE_STRUCTURE_RETAIN[3].REAL_TYPE := ARRAY_SIMPLE_STRUCTURE_RETAIN[3].REAL_TYPE + 1;
    ARRAY_SIMPLE_STRUCTURE_RETAIN[3].SINT_TYPE := ARRAY_SIMPLE_STRUCTURE_RETAIN[3].SINT_TYPE + 1;
    ARRAY_SIMPLE_STRUCTURE_RETAIN[3].STRING_TYPE := ANY_TO_STRING(ARRAY_SIMPLE_STRUCTURE_RETAIN[3].DINT_TYPE) + ' ' + ANY_TO_STRING(ARRAY_SIMPLE_STRUCTURE_RETAIN[3].TIME_TYPE);
    ARRAY_SIMPLE_STRUCTURE_RETAIN[3].TIME_TYPE := ARRAY_SIMPLE_STRUCTURE_RETAIN[3].TIME_TYPE + PULSE_TIME;
    ARRAY_SIMPLE_STRUCTURE_RETAIN[3].UDINT_TYPE := ARRAY_SIMPLE_STRUCTURE_RETAIN[3].UDINT_TYPE + 1;
    ARRAY_SIMPLE_STRUCTURE_RETAIN[3].UINT_TYPE := ARRAY_SIMPLE_STRUCTURE_RETAIN[3].UINT_TYPE + 1;
    ARRAY_SIMPLE_STRUCTURE_RETAIN[3].ULINT_TYPE := ARRAY_SIMPLE_STRUCTURE_RETAIN[3].ULINT_TYPE + 1;
    ARRAY_SIMPLE_STRUCTURE_RETAIN[3].USINT_TYPE := ARRAY_SIMPLE_STRUCTURE_RETAIN[3].USINT_TYPE + 1;
    ARRAY_SIMPLE_STRUCTURE_RETAIN[3].WORD_TYPE := ARRAY_SIMPLE_STRUCTURE_RETAIN[3].WORD_TYPE + 1;

    ARRAY_SIMPLE_STRUCTURE_RETAIN[4].BOOL_TYPE := NOT ARRAY_SIMPLE_STRUCTURE_RETAIN[4].BOOL_TYPE;
    ARRAY_SIMPLE_STRUCTURE_RETAIN[4].BYTE_TYPE := ARRAY_SIMPLE_STRUCTURE_RETAIN[4].BYTE_TYPE + 1;
    ARRAY_SIMPLE_STRUCTURE_RETAIN[4].DATE_TYPE := ANY_TO_DATE(1445385600 + ARRAY_SIMPLE_STRUCTURE_RETAIN[4].DINT_TYPE * 86400);
    ARRAY_SIMPLE_STRUCTURE_RETAIN[4].DINT_TYPE := ARRAY_SIMPLE_STRUCTURE_RETAIN[4].DINT_TYPE + 1;
    ARRAY_SIMPLE_STRUCTURE_RETAIN[4].DWORD_TYPE := ARRAY_SIMPLE_STRUCTURE_RETAIN[4].DWORD_TYPE + 1;
    ARRAY_SIMPLE_STRUCTURE_RETAIN[4].INT_TYPE := ARRAY_SIMPLE_STRUCTURE_RETAIN[4].INT_TYPE + 1;
    ARRAY_SIMPLE_STRUCTURE_RETAIN[4].LINT_TYPE := ARRAY_SIMPLE_STRUCTURE_RETAIN[4].LINT_TYPE + 1;
    ARRAY_SIMPLE_STRUCTURE_RETAIN[4].LREAL_TYPE := ARRAY_SIMPLE_STRUCTURE_RETAIN[4].LREAL_TYPE + 1;
    ARRAY_SIMPLE_STRUCTURE_RETAIN[4].LWORD_TYPE := ARRAY_SIMPLE_STRUCTURE_RETAIN[4].LWORD_TYPE + 1;
    ARRAY_SIMPLE_STRUCTURE_RETAIN[4].REAL_TYPE := ARRAY_SIMPLE_STRUCTURE_RETAIN[4].REAL_TYPE + 1;
    ARRAY_SIMPLE_STRUCTURE_RETAIN[4].SINT_TYPE := ARRAY_SIMPLE_STRUCTURE_RETAIN[4].SINT_TYPE + 1;
    ARRAY_SIMPLE_STRUCTURE_RETAIN[4].STRING_TYPE := ANY_TO_STRING(ARRAY_SIMPLE_STRUCTURE_RETAIN[4].DINT_TYPE) + ' ' + ANY_TO_STRING(ARRAY_SIMPLE_STRUCTURE_RETAIN[4].TIME_TYPE);
    ARRAY_SIMPLE_STRUCTURE_RETAIN[4].TIME_TYPE := ARRAY_SIMPLE_STRUCTURE_RETAIN[4].TIME_TYPE + PULSE_TIME;
    ARRAY_SIMPLE_STRUCTURE_RETAIN[4].UDINT_TYPE := ARRAY_SIMPLE_STRUCTURE_RETAIN[4].UDINT_TYPE + 1;
    ARRAY_SIMPLE_STRUCTURE_RETAIN[4].UINT_TYPE := ARRAY_SIMPLE_STRUCTURE_RETAIN[4].UINT_TYPE + 1;
    ARRAY_SIMPLE_STRUCTURE_RETAIN[4].ULINT_TYPE := ARRAY_SIMPLE_STRUCTURE_RETAIN[4].ULINT_TYPE + 1;
    ARRAY_SIMPLE_STRUCTURE_RETAIN[4].USINT_TYPE := ARRAY_SIMPLE_STRUCTURE_RETAIN[4].USINT_TYPE + 1;
    ARRAY_SIMPLE_STRUCTURE_RETAIN[4].WORD_TYPE := ARRAY_SIMPLE_STRUCTURE_RETAIN[4].WORD_TYPE + 1;

    ARRAY_SIMPLE_STRUCTURE_RETAIN[5].BOOL_TYPE := ARRAY_SIMPLE_STRUCTURE_RETAIN[4].BOOL_TYPE;
    ARRAY_SIMPLE_STRUCTURE_RETAIN[5].BYTE_TYPE := ARRAY_SIMPLE_STRUCTURE_RETAIN[4].BYTE_TYPE;
    ARRAY_SIMPLE_STRUCTURE_RETAIN[5].DATE_TYPE := ARRAY_SIMPLE_STRUCTURE_RETAIN[4].DATE_TYPE;
    ARRAY_SIMPLE_STRUCTURE_RETAIN[5].DINT_TYPE := ARRAY_SIMPLE_STRUCTURE_RETAIN[4].DINT_TYPE;
    ARRAY_SIMPLE_STRUCTURE_RETAIN[5].DWORD_TYPE := ARRAY_SIMPLE_STRUCTURE_RETAIN[4].DWORD_TYPE;
    ARRAY_SIMPLE_STRUCTURE_RETAIN[5].INT_TYPE := ARRAY_SIMPLE_STRUCTURE_RETAIN[4].INT_TYPE;
    ARRAY_SIMPLE_STRUCTURE_RETAIN[5].LINT_TYPE := ARRAY_SIMPLE_STRUCTURE_RETAIN[4].LINT_TYPE;
    ARRAY_SIMPLE_STRUCTURE_RETAIN[5].LREAL_TYPE := ARRAY_SIMPLE_STRUCTURE_RETAIN[4].LREAL_TYPE;
    ARRAY_SIMPLE_STRUCTURE_RETAIN[5].LWORD_TYPE := ARRAY_SIMPLE_STRUCTURE_RETAIN[4].LWORD_TYPE;
    ARRAY_SIMPLE_STRUCTURE_RETAIN[5].REAL_TYPE := ARRAY_SIMPLE_STRUCTURE_RETAIN[4].REAL_TYPE;
    ARRAY_SIMPLE_STRUCTURE_RETAIN[5].SINT_TYPE := ARRAY_SIMPLE_STRUCTURE_RETAIN[4].SINT_TYPE;
    ARRAY_SIMPLE_STRUCTURE_RETAIN[5].STRING_TYPE := ARRAY_SIMPLE_STRUCTURE_RETAIN[4].STRING_TYPE;
    ARRAY_SIMPLE_STRUCTURE_RETAIN[5].TIME_TYPE := ARRAY_SIMPLE_STRUCTURE_RETAIN[4].TIME_TYPE;
    ARRAY_SIMPLE_STRUCTURE_RETAIN[5].UDINT_TYPE := ARRAY_SIMPLE_STRUCTURE_RETAIN[4].UDINT_TYPE;
    ARRAY_SIMPLE_STRUCTURE_RETAIN[5].UINT_TYPE := ARRAY_SIMPLE_STRUCTURE_RETAIN[4].UINT_TYPE;
    ARRAY_SIMPLE_STRUCTURE_RETAIN[5].ULINT_TYPE := ARRAY_SIMPLE_STRUCTURE_RETAIN[4].ULINT_TYPE;
    ARRAY_SIMPLE_STRUCTURE_RETAIN[5].USINT_TYPE := ARRAY_SIMPLE_STRUCTURE_RETAIN[4].USINT_TYPE;
    ARRAY_SIMPLE_STRUCTURE_RETAIN[5].WORD_TYPE := ARRAY_SIMPLE_STRUCTURE_RETAIN[4].WORD_TYPE;

    ARRAY_SIMPLE_STRUCTURE_NON_RETAIN[0].BOOL_TYPE := NOT ARRAY_SIMPLE_STRUCTURE_NON_RETAIN[0].BOOL_TYPE;
    ARRAY_SIMPLE_STRUCTURE_NON_RETAIN[0].BYTE_TYPE := ARRAY_SIMPLE_STRUCTURE_NON_RETAIN[0].BYTE_TYPE + 1;
    ARRAY_SIMPLE_STRUCTURE_NON_RETAIN[0].DATE_TYPE := ANY_TO_DATE(1445385600 + ARRAY_SIMPLE_STRUCTURE_NON_RETAIN[0].DINT_TYPE * 86400);
    ARRAY_SIMPLE_STRUCTURE_NON_RETAIN[0].DINT_TYPE := ARRAY_SIMPLE_STRUCTURE_NON_RETAIN[0].DINT_TYPE + 1;
    ARRAY_SIMPLE_STRUCTURE_NON_RETAIN[0].DWORD_TYPE := ARRAY_SIMPLE_STRUCTURE_NON_RETAIN[0].DWORD_TYPE + 1;
    ARRAY_SIMPLE_STRUCTURE_NON_RETAIN[0].INT_TYPE := ARRAY_SIMPLE_STRUCTURE_NON_RETAIN[0].INT_TYPE + 1;
    ARRAY_SIMPLE_STRUCTURE_NON_RETAIN[0].LINT_TYPE := ARRAY_SIMPLE_STRUCTURE_NON_RETAIN[0].LINT_TYPE + 1;
    ARRAY_SIMPLE_STRUCTURE_NON_RETAIN[0].LREAL_TYPE := ARRAY_SIMPLE_STRUCTURE_NON_RETAIN[0].LREAL_TYPE + 1;
    ARRAY_SIMPLE_STRUCTURE_NON_RETAIN[0].LWORD_TYPE := ARRAY_SIMPLE_STRUCTURE_NON_RETAIN[0].LWORD_TYPE + 1;
    ARRAY_SIMPLE_STRUCTURE_NON_RETAIN[0].REAL_TYPE := ARRAY_SIMPLE_STRUCTURE_NON_RETAIN[0].REAL_TYPE + 1;
    ARRAY_SIMPLE_STRUCTURE_NON_RETAIN[0].SINT_TYPE := ARRAY_SIMPLE_STRUCTURE_NON_RETAIN[0].SINT_TYPE + 1;
    ARRAY_SIMPLE_STRUCTURE_NON_RETAIN[0].STRING_TYPE := ANY_TO_STRING(ARRAY_SIMPLE_STRUCTURE_NON_RETAIN[0].DINT_TYPE) + ' ' + ANY_TO_STRING(ARRAY_SIMPLE_STRUCTURE_NON_RETAIN[0].TIME_TYPE);
    ARRAY_SIMPLE_STRUCTURE_NON_RETAIN[0].TIME_TYPE := ARRAY_SIMPLE_STRUCTURE_NON_RETAIN[0].TIME_TYPE + PULSE_TIME;
    ARRAY_SIMPLE_STRUCTURE_NON_RETAIN[0].UDINT_TYPE := ARRAY_SIMPLE_STRUCTURE_NON_RETAIN[0].UDINT_TYPE + 1;
    ARRAY_SIMPLE_STRUCTURE_NON_RETAIN[0].UINT_TYPE := ARRAY_SIMPLE_STRUCTURE_NON_RETAIN[0].UINT_TYPE + 1;
    ARRAY_SIMPLE_STRUCTURE_NON_RETAIN[0].ULINT_TYPE := ARRAY_SIMPLE_STRUCTURE_NON_RETAIN[0].ULINT_TYPE + 1;
    ARRAY_SIMPLE_STRUCTURE_NON_RETAIN[0].USINT_TYPE := ARRAY_SIMPLE_STRUCTURE_NON_RETAIN[0].USINT_TYPE + 1;
    ARRAY_SIMPLE_STRUCTURE_NON_RETAIN[0].WORD_TYPE := ARRAY_SIMPLE_STRUCTURE_NON_RETAIN[0].WORD_TYPE + 1;

    ARRAY_SIMPLE_STRUCTURE_NON_RETAIN[1].BOOL_TYPE := NOT ARRAY_SIMPLE_STRUCTURE_NON_RETAIN[1].BOOL_TYPE;
    ARRAY_SIMPLE_STRUCTURE_NON_RETAIN[1].BYTE_TYPE := ARRAY_SIMPLE_STRUCTURE_NON_RETAIN[1].BYTE_TYPE + 1;
    ARRAY_SIMPLE_STRUCTURE_NON_RETAIN[1].DATE_TYPE := ANY_TO_DATE(1445385600 + ARRAY_SIMPLE_STRUCTURE_NON_RETAIN[1].DINT_TYPE * 86400);
    ARRAY_SIMPLE_STRUCTURE_NON_RETAIN[1].DINT_TYPE := ARRAY_SIMPLE_STRUCTURE_NON_RETAIN[1].DINT_TYPE + 1;
    ARRAY_SIMPLE_STRUCTURE_NON_RETAIN[1].DWORD_TYPE := ARRAY_SIMPLE_STRUCTURE_NON_RETAIN[1].DWORD_TYPE + 1;
    ARRAY_SIMPLE_STRUCTURE_NON_RETAIN[1].INT_TYPE := ARRAY_SIMPLE_STRUCTURE_NON_RETAIN[1].INT_TYPE + 1;
    ARRAY_SIMPLE_STRUCTURE_NON_RETAIN[1].LINT_TYPE := ARRAY_SIMPLE_STRUCTURE_NON_RETAIN[1].LINT_TYPE + 1;
    ARRAY_SIMPLE_STRUCTURE_NON_RETAIN[1].LREAL_TYPE := ARRAY_SIMPLE_STRUCTURE_NON_RETAIN[1].LREAL_TYPE + 1;
    ARRAY_SIMPLE_STRUCTURE_NON_RETAIN[1].LWORD_TYPE := ARRAY_SIMPLE_STRUCTURE_NON_RETAIN[1].LWORD_TYPE + 1;
    ARRAY_SIMPLE_STRUCTURE_NON_RETAIN[1].REAL_TYPE := ARRAY_SIMPLE_STRUCTURE_NON_RETAIN[1].REAL_TYPE + 1;
    ARRAY_SIMPLE_STRUCTURE_NON_RETAIN[1].SINT_TYPE := ARRAY_SIMPLE_STRUCTURE_NON_RETAIN[1].SINT_TYPE + 1;
    ARRAY_SIMPLE_STRUCTURE_NON_RETAIN[1].STRING_TYPE := ANY_TO_STRING(ARRAY_SIMPLE_STRUCTURE_NON_RETAIN[1].DINT_TYPE) + ' ' + ANY_TO_STRING(ARRAY_SIMPLE_STRUCTURE_NON_RETAIN[1].TIME_TYPE);
    ARRAY_SIMPLE_STRUCTURE_NON_RETAIN[1].TIME_TYPE := ARRAY_SIMPLE_STRUCTURE_NON_RETAIN[1].TIME_TYPE + PULSE_TIME;
    ARRAY_SIMPLE_STRUCTURE_NON_RETAIN[1].UDINT_TYPE := ARRAY_SIMPLE_STRUCTURE_NON_RETAIN[1].UDINT_TYPE + 1;
    ARRAY_SIMPLE_STRUCTURE_NON_RETAIN[1].UINT_TYPE := ARRAY_SIMPLE_STRUCTURE_NON_RETAIN[1].UINT_TYPE + 1;
    ARRAY_SIMPLE_STRUCTURE_NON_RETAIN[1].ULINT_TYPE := ARRAY_SIMPLE_STRUCTURE_NON_RETAIN[1].ULINT_TYPE + 1;
    ARRAY_SIMPLE_STRUCTURE_NON_RETAIN[1].USINT_TYPE := ARRAY_SIMPLE_STRUCTURE_NON_RETAIN[1].USINT_TYPE + 1;
    ARRAY_SIMPLE_STRUCTURE_NON_RETAIN[1].WORD_TYPE := ARRAY_SIMPLE_STRUCTURE_NON_RETAIN[1].WORD_TYPE + 1;

    ARRAY_SIMPLE_STRUCTURE_NON_RETAIN[2].BOOL_TYPE := NOT ARRAY_SIMPLE_STRUCTURE_NON_RETAIN[2].BOOL_TYPE;
    ARRAY_SIMPLE_STRUCTURE_NON_RETAIN[2].BYTE_TYPE := ARRAY_SIMPLE_STRUCTURE_NON_RETAIN[2].BYTE_TYPE + 1;
    ARRAY_SIMPLE_STRUCTURE_NON_RETAIN[2].DATE_TYPE := ANY_TO_DATE(1445385600 + ARRAY_SIMPLE_STRUCTURE_NON_RETAIN[2].DINT_TYPE * 86400);
    ARRAY_SIMPLE_STRUCTURE_NON_RETAIN[2].DINT_TYPE := ARRAY_SIMPLE_STRUCTURE_NON_RETAIN[2].DINT_TYPE + 1;
    ARRAY_SIMPLE_STRUCTURE_NON_RETAIN[2].DWORD_TYPE := ARRAY_SIMPLE_STRUCTURE_NON_RETAIN[2].DWORD_TYPE + 1;
    ARRAY_SIMPLE_STRUCTURE_NON_RETAIN[2].INT_TYPE := ARRAY_SIMPLE_STRUCTURE_NON_RETAIN[2].INT_TYPE + 1;
    ARRAY_SIMPLE_STRUCTURE_NON_RETAIN[2].LINT_TYPE := ARRAY_SIMPLE_STRUCTURE_NON_RETAIN[2].LINT_TYPE + 1;
    ARRAY_SIMPLE_STRUCTURE_NON_RETAIN[2].LREAL_TYPE := ARRAY_SIMPLE_STRUCTURE_NON_RETAIN[2].LREAL_TYPE + 1;
    ARRAY_SIMPLE_STRUCTURE_NON_RETAIN[2].LWORD_TYPE := ARRAY_SIMPLE_STRUCTURE_NON_RETAIN[2].LWORD_TYPE + 1;
    ARRAY_SIMPLE_STRUCTURE_NON_RETAIN[2].REAL_TYPE := ARRAY_SIMPLE_STRUCTURE_NON_RETAIN[2].REAL_TYPE + 1;
    ARRAY_SIMPLE_STRUCTURE_NON_RETAIN[2].SINT_TYPE := ARRAY_SIMPLE_STRUCTURE_NON_RETAIN[2].SINT_TYPE + 1;
    ARRAY_SIMPLE_STRUCTURE_NON_RETAIN[2].STRING_TYPE := ANY_TO_STRING(ARRAY_SIMPLE_STRUCTURE_NON_RETAIN[2].DINT_TYPE) + ' ' + ANY_TO_STRING(ARRAY_SIMPLE_STRUCTURE_NON_RETAIN[2].TIME_TYPE);
    ARRAY_SIMPLE_STRUCTURE_NON_RETAIN[2].TIME_TYPE := ARRAY_SIMPLE_STRUCTURE_NON_RETAIN[2].TIME_TYPE + PULSE_TIME;
    ARRAY_SIMPLE_STRUCTURE_NON_RETAIN[2].UDINT_TYPE := ARRAY_SIMPLE_STRUCTURE_NON_RETAIN[2].UDINT_TYPE + 1;
    ARRAY_SIMPLE_STRUCTURE_NON_RETAIN[2].UINT_TYPE := ARRAY_SIMPLE_STRUCTURE_NON_RETAIN[2].UINT_TYPE + 1;
    ARRAY_SIMPLE_STRUCTURE_NON_RETAIN[2].ULINT_TYPE := ARRAY_SIMPLE_STRUCTURE_NON_RETAIN[2].ULINT_TYPE + 1;
    ARRAY_SIMPLE_STRUCTURE_NON_RETAIN[2].USINT_TYPE := ARRAY_SIMPLE_STRUCTURE_NON_RETAIN[2].USINT_TYPE + 1;
    ARRAY_SIMPLE_STRUCTURE_NON_RETAIN[2].WORD_TYPE := ARRAY_SIMPLE_STRUCTURE_NON_RETAIN[2].WORD_TYPE + 1;

    ARRAY_SIMPLE_STRUCTURE_NON_RETAIN[3].BOOL_TYPE := NOT ARRAY_SIMPLE_STRUCTURE_NON_RETAIN[3].BOOL_TYPE;
    ARRAY_SIMPLE_STRUCTURE_NON_RETAIN[3].BYTE_TYPE := ARRAY_SIMPLE_STRUCTURE_NON_RETAIN[3].BYTE_TYPE + 1;
    ARRAY_SIMPLE_STRUCTURE_NON_RETAIN[3].DATE_TYPE := ANY_TO_DATE(1445385600 + ARRAY_SIMPLE_STRUCTURE_NON_RETAIN[3].DINT_TYPE * 86400);
    ARRAY_SIMPLE_STRUCTURE_NON_RETAIN[3].DINT_TYPE := ARRAY_SIMPLE_STRUCTURE_NON_RETAIN[3].DINT_TYPE + 1;
    ARRAY_SIMPLE_STRUCTURE_NON_RETAIN[3].DWORD_TYPE := ARRAY_SIMPLE_STRUCTURE_NON_RETAIN[3].DWORD_TYPE + 1;
    ARRAY_SIMPLE_STRUCTURE_NON_RETAIN[3].INT_TYPE := ARRAY_SIMPLE_STRUCTURE_NON_RETAIN[3].INT_TYPE + 1;
    ARRAY_SIMPLE_STRUCTURE_NON_RETAIN[3].LINT_TYPE := ARRAY_SIMPLE_STRUCTURE_NON_RETAIN[3].LINT_TYPE + 1;
    ARRAY_SIMPLE_STRUCTURE_NON_RETAIN[3].LREAL_TYPE := ARRAY_SIMPLE_STRUCTURE_NON_RETAIN[3].LREAL_TYPE + 1;
    ARRAY_SIMPLE_STRUCTURE_NON_RETAIN[3].LWORD_TYPE := ARRAY_SIMPLE_STRUCTURE_NON_RETAIN[3].LWORD_TYPE + 1;
    ARRAY_SIMPLE_STRUCTURE_NON_RETAIN[3].REAL_TYPE := ARRAY_SIMPLE_STRUCTURE_NON_RETAIN[3].REAL_TYPE + 1;
    ARRAY_SIMPLE_STRUCTURE_NON_RETAIN[3].SINT_TYPE := ARRAY_SIMPLE_STRUCTURE_NON_RETAIN[3].SINT_TYPE + 1;
    ARRAY_SIMPLE_STRUCTURE_NON_RETAIN[3].STRING_TYPE := ANY_TO_STRING(ARRAY_SIMPLE_STRUCTURE_NON_RETAIN[3].DINT_TYPE) + ' ' + ANY_TO_STRING(ARRAY_SIMPLE_STRUCTURE_NON_RETAIN[3].TIME_TYPE);
    ARRAY_SIMPLE_STRUCTURE_NON_RETAIN[3].TIME_TYPE := ARRAY_SIMPLE_STRUCTURE_NON_RETAIN[3].TIME_TYPE + PULSE_TIME;
    ARRAY_SIMPLE_STRUCTURE_NON_RETAIN[3].UDINT_TYPE := ARRAY_SIMPLE_STRUCTURE_NON_RETAIN[3].UDINT_TYPE + 1;
    ARRAY_SIMPLE_STRUCTURE_NON_RETAIN[3].UINT_TYPE := ARRAY_SIMPLE_STRUCTURE_NON_RETAIN[3].UINT_TYPE + 1;
    ARRAY_SIMPLE_STRUCTURE_NON_RETAIN[3].ULINT_TYPE := ARRAY_SIMPLE_STRUCTURE_NON_RETAIN[3].ULINT_TYPE + 1;
    ARRAY_SIMPLE_STRUCTURE_NON_RETAIN[3].USINT_TYPE := ARRAY_SIMPLE_STRUCTURE_NON_RETAIN[3].USINT_TYPE + 1;
    ARRAY_SIMPLE_STRUCTURE_NON_RETAIN[3].WORD_TYPE := ARRAY_SIMPLE_STRUCTURE_NON_RETAIN[3].WORD_TYPE + 1;

    ARRAY_SIMPLE_STRUCTURE_NON_RETAIN[4].BOOL_TYPE := NOT ARRAY_SIMPLE_STRUCTURE_NON_RETAIN[4].BOOL_TYPE;
    ARRAY_SIMPLE_STRUCTURE_NON_RETAIN[4].BYTE_TYPE := ARRAY_SIMPLE_STRUCTURE_NON_RETAIN[4].BYTE_TYPE + 1;
    ARRAY_SIMPLE_STRUCTURE_NON_RETAIN[4].DATE_TYPE := ANY_TO_DATE(1445385600 + ARRAY_SIMPLE_STRUCTURE_NON_RETAIN[4].DINT_TYPE * 86400);
    ARRAY_SIMPLE_STRUCTURE_NON_RETAIN[4].DINT_TYPE := ARRAY_SIMPLE_STRUCTURE_NON_RETAIN[4].DINT_TYPE + 1;
    ARRAY_SIMPLE_STRUCTURE_NON_RETAIN[4].DWORD_TYPE := ARRAY_SIMPLE_STRUCTURE_NON_RETAIN[4].DWORD_TYPE + 1;
    ARRAY_SIMPLE_STRUCTURE_NON_RETAIN[4].INT_TYPE := ARRAY_SIMPLE_STRUCTURE_NON_RETAIN[4].INT_TYPE + 1;
    ARRAY_SIMPLE_STRUCTURE_NON_RETAIN[4].LINT_TYPE := ARRAY_SIMPLE_STRUCTURE_NON_RETAIN[4].LINT_TYPE + 1;
    ARRAY_SIMPLE_STRUCTURE_NON_RETAIN[4].LREAL_TYPE := ARRAY_SIMPLE_STRUCTURE_NON_RETAIN[4].LREAL_TYPE + 1;
    ARRAY_SIMPLE_STRUCTURE_NON_RETAIN[4].LWORD_TYPE := ARRAY_SIMPLE_STRUCTURE_NON_RETAIN[4].LWORD_TYPE + 1;
    ARRAY_SIMPLE_STRUCTURE_NON_RETAIN[4].REAL_TYPE := ARRAY_SIMPLE_STRUCTURE_NON_RETAIN[4].REAL_TYPE + 1;
    ARRAY_SIMPLE_STRUCTURE_NON_RETAIN[4].SINT_TYPE := ARRAY_SIMPLE_STRUCTURE_NON_RETAIN[4].SINT_TYPE + 1;
    ARRAY_SIMPLE_STRUCTURE_NON_RETAIN[4].STRING_TYPE := ANY_TO_STRING(ARRAY_SIMPLE_STRUCTURE_NON_RETAIN[4].DINT_TYPE) + ' ' + ANY_TO_STRING(ARRAY_SIMPLE_STRUCTURE_NON_RETAIN[4].TIME_TYPE);
    ARRAY_SIMPLE_STRUCTURE_NON_RETAIN[4].TIME_TYPE := ARRAY_SIMPLE_STRUCTURE_NON_RETAIN[4].TIME_TYPE + PULSE_TIME;
    ARRAY_SIMPLE_STRUCTURE_NON_RETAIN[4].UDINT_TYPE := ARRAY_SIMPLE_STRUCTURE_NON_RETAIN[4].UDINT_TYPE + 1;
    ARRAY_SIMPLE_STRUCTURE_NON_RETAIN[4].UINT_TYPE := ARRAY_SIMPLE_STRUCTURE_NON_RETAIN[4].UINT_TYPE + 1;
    ARRAY_SIMPLE_STRUCTURE_NON_RETAIN[4].ULINT_TYPE := ARRAY_SIMPLE_STRUCTURE_NON_RETAIN[4].ULINT_TYPE + 1;
    ARRAY_SIMPLE_STRUCTURE_NON_RETAIN[4].USINT_TYPE := ARRAY_SIMPLE_STRUCTURE_NON_RETAIN[4].USINT_TYPE + 1;
    ARRAY_SIMPLE_STRUCTURE_NON_RETAIN[4].WORD_TYPE := ARRAY_SIMPLE_STRUCTURE_NON_RETAIN[4].WORD_TYPE + 1;

    ARRAY_SIMPLE_STRUCTURE_NON_RETAIN[5].BOOL_TYPE := ARRAY_SIMPLE_STRUCTURE_NON_RETAIN[4].BOOL_TYPE;
    ARRAY_SIMPLE_STRUCTURE_NON_RETAIN[5].BYTE_TYPE := ARRAY_SIMPLE_STRUCTURE_NON_RETAIN[4].BYTE_TYPE;
    ARRAY_SIMPLE_STRUCTURE_NON_RETAIN[5].DATE_TYPE := ARRAY_SIMPLE_STRUCTURE_NON_RETAIN[4].DATE_TYPE;
    ARRAY_SIMPLE_STRUCTURE_NON_RETAIN[5].DINT_TYPE := ARRAY_SIMPLE_STRUCTURE_NON_RETAIN[4].DINT_TYPE;
    ARRAY_SIMPLE_STRUCTURE_NON_RETAIN[5].DWORD_TYPE := ARRAY_SIMPLE_STRUCTURE_NON_RETAIN[4].DWORD_TYPE;
    ARRAY_SIMPLE_STRUCTURE_NON_RETAIN[5].INT_TYPE := ARRAY_SIMPLE_STRUCTURE_NON_RETAIN[4].INT_TYPE;
    ARRAY_SIMPLE_STRUCTURE_NON_RETAIN[5].LINT_TYPE := ARRAY_SIMPLE_STRUCTURE_NON_RETAIN[4].LINT_TYPE;
    ARRAY_SIMPLE_STRUCTURE_NON_RETAIN[5].LREAL_TYPE := ARRAY_SIMPLE_STRUCTURE_NON_RETAIN[4].LREAL_TYPE;
    ARRAY_SIMPLE_STRUCTURE_NON_RETAIN[5].LWORD_TYPE := ARRAY_SIMPLE_STRUCTURE_NON_RETAIN[4].LWORD_TYPE;
    ARRAY_SIMPLE_STRUCTURE_NON_RETAIN[5].REAL_TYPE := ARRAY_SIMPLE_STRUCTURE_NON_RETAIN[4].REAL_TYPE;
    ARRAY_SIMPLE_STRUCTURE_NON_RETAIN[5].SINT_TYPE := ARRAY_SIMPLE_STRUCTURE_NON_RETAIN[4].SINT_TYPE;
    ARRAY_SIMPLE_STRUCTURE_NON_RETAIN[5].STRING_TYPE := ARRAY_SIMPLE_STRUCTURE_NON_RETAIN[4].STRING_TYPE;
    ARRAY_SIMPLE_STRUCTURE_NON_RETAIN[5].TIME_TYPE := ARRAY_SIMPLE_STRUCTURE_NON_RETAIN[4].TIME_TYPE;
    ARRAY_SIMPLE_STRUCTURE_NON_RETAIN[5].UDINT_TYPE := ARRAY_SIMPLE_STRUCTURE_NON_RETAIN[4].UDINT_TYPE;
    ARRAY_SIMPLE_STRUCTURE_NON_RETAIN[5].UINT_TYPE := ARRAY_SIMPLE_STRUCTURE_NON_RETAIN[4].UINT_TYPE;
    ARRAY_SIMPLE_STRUCTURE_NON_RETAIN[5].ULINT_TYPE := ARRAY_SIMPLE_STRUCTURE_NON_RETAIN[4].ULINT_TYPE;
    ARRAY_SIMPLE_STRUCTURE_NON_RETAIN[5].USINT_TYPE := ARRAY_SIMPLE_STRUCTURE_NON_RETAIN[4].USINT_TYPE;
    ARRAY_SIMPLE_STRUCTURE_NON_RETAIN[5].WORD_TYPE := ARRAY_SIMPLE_STRUCTURE_NON_RETAIN[4].WORD_TYPE;

    ARRAY_SIMPLE_STRUCTURE_AUTO[0].BOOL_TYPE := NOT ARRAY_SIMPLE_STRUCTURE_AUTO[0].BOOL_TYPE;
    ARRAY_SIMPLE_STRUCTURE_AUTO[0].BYTE_TYPE := ARRAY_SIMPLE_STRUCTURE_AUTO[0].BYTE_TYPE + 1;
    ARRAY_SIMPLE_STRUCTURE_AUTO[0].DATE_TYPE := ANY_TO_DATE(1445385600 + ARRAY_SIMPLE_STRUCTURE_AUTO[0].DINT_TYPE * 86400);
    ARRAY_SIMPLE_STRUCTURE_AUTO[0].DINT_TYPE := ARRAY_SIMPLE_STRUCTURE_AUTO[0].DINT_TYPE + 1;
    ARRAY_SIMPLE_STRUCTURE_AUTO[0].DWORD_TYPE := ARRAY_SIMPLE_STRUCTURE_AUTO[0].DWORD_TYPE + 1;
    ARRAY_SIMPLE_STRUCTURE_AUTO[0].INT_TYPE := ARRAY_SIMPLE_STRUCTURE_AUTO[0].INT_TYPE + 1;
    ARRAY_SIMPLE_STRUCTURE_AUTO[0].LINT_TYPE := ARRAY_SIMPLE_STRUCTURE_AUTO[0].LINT_TYPE + 1;
    ARRAY_SIMPLE_STRUCTURE_AUTO[0].LREAL_TYPE := ARRAY_SIMPLE_STRUCTURE_AUTO[0].LREAL_TYPE + 1;
    ARRAY_SIMPLE_STRUCTURE_AUTO[0].LWORD_TYPE := ARRAY_SIMPLE_STRUCTURE_AUTO[0].LWORD_TYPE + 1;
    ARRAY_SIMPLE_STRUCTURE_AUTO[0].REAL_TYPE := ARRAY_SIMPLE_STRUCTURE_AUTO[0].REAL_TYPE + 1;
    ARRAY_SIMPLE_STRUCTURE_AUTO[0].SINT_TYPE := ARRAY_SIMPLE_STRUCTURE_AUTO[0].SINT_TYPE + 1;
    ARRAY_SIMPLE_STRUCTURE_AUTO[0].STRING_TYPE := ANY_TO_STRING(ARRAY_SIMPLE_STRUCTURE_AUTO[0].DINT_TYPE) + ' ' + ANY_TO_STRING(ARRAY_SIMPLE_STRUCTURE_AUTO[0].TIME_TYPE);
    ARRAY_SIMPLE_STRUCTURE_AUTO[0].TIME_TYPE := ARRAY_SIMPLE_STRUCTURE_AUTO[0].TIME_TYPE + PULSE_TIME;
    ARRAY_SIMPLE_STRUCTURE_AUTO[0].UDINT_TYPE := ARRAY_SIMPLE_STRUCTURE_AUTO[0].UDINT_TYPE + 1;
    ARRAY_SIMPLE_STRUCTURE_AUTO[0].UINT_TYPE := ARRAY_SIMPLE_STRUCTURE_AUTO[0].UINT_TYPE + 1;
    ARRAY_SIMPLE_STRUCTURE_AUTO[0].ULINT_TYPE := ARRAY_SIMPLE_STRUCTURE_AUTO[0].ULINT_TYPE + 1;
    ARRAY_SIMPLE_STRUCTURE_AUTO[0].USINT_TYPE := ARRAY_SIMPLE_STRUCTURE_AUTO[0].USINT_TYPE + 1;
    ARRAY_SIMPLE_STRUCTURE_AUTO[0].WORD_TYPE := ARRAY_SIMPLE_STRUCTURE_AUTO[0].WORD_TYPE + 1;

    ARRAY_SIMPLE_STRUCTURE_AUTO[1].BOOL_TYPE := NOT ARRAY_SIMPLE_STRUCTURE_AUTO[1].BOOL_TYPE;
    ARRAY_SIMPLE_STRUCTURE_AUTO[1].BYTE_TYPE := ARRAY_SIMPLE_STRUCTURE_AUTO[1].BYTE_TYPE + 1;
    ARRAY_SIMPLE_STRUCTURE_AUTO[1].DATE_TYPE := ANY_TO_DATE(1445385600 + ARRAY_SIMPLE_STRUCTURE_AUTO[1].DINT_TYPE * 86400);
    ARRAY_SIMPLE_STRUCTURE_AUTO[1].DINT_TYPE := ARRAY_SIMPLE_STRUCTURE_AUTO[1].DINT_TYPE + 1;
    ARRAY_SIMPLE_STRUCTURE_AUTO[1].DWORD_TYPE := ARRAY_SIMPLE_STRUCTURE_AUTO[1].DWORD_TYPE + 1;
    ARRAY_SIMPLE_STRUCTURE_AUTO[1].INT_TYPE := ARRAY_SIMPLE_STRUCTURE_AUTO[1].INT_TYPE + 1;
    ARRAY_SIMPLE_STRUCTURE_AUTO[1].LINT_TYPE := ARRAY_SIMPLE_STRUCTURE_AUTO[1].LINT_TYPE + 1;
    ARRAY_SIMPLE_STRUCTURE_AUTO[1].LREAL_TYPE := ARRAY_SIMPLE_STRUCTURE_AUTO[1].LREAL_TYPE + 1;
    ARRAY_SIMPLE_STRUCTURE_AUTO[1].LWORD_TYPE := ARRAY_SIMPLE_STRUCTURE_AUTO[1].LWORD_TYPE + 1;
    ARRAY_SIMPLE_STRUCTURE_AUTO[1].REAL_TYPE := ARRAY_SIMPLE_STRUCTURE_AUTO[1].REAL_TYPE + 1;
    ARRAY_SIMPLE_STRUCTURE_AUTO[1].SINT_TYPE := ARRAY_SIMPLE_STRUCTURE_AUTO[1].SINT_TYPE + 1;
    ARRAY_SIMPLE_STRUCTURE_AUTO[1].STRING_TYPE := ANY_TO_STRING(ARRAY_SIMPLE_STRUCTURE_AUTO[1].DINT_TYPE) + ' ' + ANY_TO_STRING(ARRAY_SIMPLE_STRUCTURE_AUTO[1].TIME_TYPE);
    ARRAY_SIMPLE_STRUCTURE_AUTO[1].TIME_TYPE := ARRAY_SIMPLE_STRUCTURE_AUTO[1].TIME_TYPE + PULSE_TIME;
    ARRAY_SIMPLE_STRUCTURE_AUTO[1].UDINT_TYPE := ARRAY_SIMPLE_STRUCTURE_AUTO[1].UDINT_TYPE + 1;
    ARRAY_SIMPLE_STRUCTURE_AUTO[1].UINT_TYPE := ARRAY_SIMPLE_STRUCTURE_AUTO[1].UINT_TYPE + 1;
    ARRAY_SIMPLE_STRUCTURE_AUTO[1].ULINT_TYPE := ARRAY_SIMPLE_STRUCTURE_AUTO[1].ULINT_TYPE + 1;
    ARRAY_SIMPLE_STRUCTURE_AUTO[1].USINT_TYPE := ARRAY_SIMPLE_STRUCTURE_AUTO[1].USINT_TYPE + 1;
    ARRAY_SIMPLE_STRUCTURE_AUTO[1].WORD_TYPE := ARRAY_SIMPLE_STRUCTURE_AUTO[1].WORD_TYPE + 1;

    ARRAY_SIMPLE_STRUCTURE_AUTO[2].BOOL_TYPE := NOT ARRAY_SIMPLE_STRUCTURE_AUTO[2].BOOL_TYPE;
    ARRAY_SIMPLE_STRUCTURE_AUTO[2].BYTE_TYPE := ARRAY_SIMPLE_STRUCTURE_AUTO[2].BYTE_TYPE + 1;
    ARRAY_SIMPLE_STRUCTURE_AUTO[2].DATE_TYPE := ANY_TO_DATE(1445385600 + ARRAY_SIMPLE_STRUCTURE_AUTO[2].DINT_TYPE * 86400);
    ARRAY_SIMPLE_STRUCTURE_AUTO[2].DINT_TYPE := ARRAY_SIMPLE_STRUCTURE_AUTO[2].DINT_TYPE + 1;
    ARRAY_SIMPLE_STRUCTURE_AUTO[2].DWORD_TYPE := ARRAY_SIMPLE_STRUCTURE_AUTO[2].DWORD_TYPE + 1;
    ARRAY_SIMPLE_STRUCTURE_AUTO[2].INT_TYPE := ARRAY_SIMPLE_STRUCTURE_AUTO[2].INT_TYPE + 1;
    ARRAY_SIMPLE_STRUCTURE_AUTO[2].LINT_TYPE := ARRAY_SIMPLE_STRUCTURE_AUTO[2].LINT_TYPE + 1;
    ARRAY_SIMPLE_STRUCTURE_AUTO[2].LREAL_TYPE := ARRAY_SIMPLE_STRUCTURE_AUTO[2].LREAL_TYPE + 1;
    ARRAY_SIMPLE_STRUCTURE_AUTO[2].LWORD_TYPE := ARRAY_SIMPLE_STRUCTURE_AUTO[2].LWORD_TYPE + 1;
    ARRAY_SIMPLE_STRUCTURE_AUTO[2].REAL_TYPE := ARRAY_SIMPLE_STRUCTURE_AUTO[2].REAL_TYPE + 1;
    ARRAY_SIMPLE_STRUCTURE_AUTO[2].SINT_TYPE := ARRAY_SIMPLE_STRUCTURE_AUTO[2].SINT_TYPE + 1;
    ARRAY_SIMPLE_STRUCTURE_AUTO[2].STRING_TYPE := ANY_TO_STRING(ARRAY_SIMPLE_STRUCTURE_AUTO[2].DINT_TYPE) + ' ' + ANY_TO_STRING(ARRAY_SIMPLE_STRUCTURE_AUTO[2].TIME_TYPE);
    ARRAY_SIMPLE_STRUCTURE_AUTO[2].TIME_TYPE := ARRAY_SIMPLE_STRUCTURE_AUTO[2].TIME_TYPE + PULSE_TIME;
    ARRAY_SIMPLE_STRUCTURE_AUTO[2].UDINT_TYPE := ARRAY_SIMPLE_STRUCTURE_AUTO[2].UDINT_TYPE + 1;
    ARRAY_SIMPLE_STRUCTURE_AUTO[2].UINT_TYPE := ARRAY_SIMPLE_STRUCTURE_AUTO[2].UINT_TYPE + 1;
    ARRAY_SIMPLE_STRUCTURE_AUTO[2].ULINT_TYPE := ARRAY_SIMPLE_STRUCTURE_AUTO[2].ULINT_TYPE + 1;
    ARRAY_SIMPLE_STRUCTURE_AUTO[2].USINT_TYPE := ARRAY_SIMPLE_STRUCTURE_AUTO[2].USINT_TYPE + 1;
    ARRAY_SIMPLE_STRUCTURE_AUTO[2].WORD_TYPE := ARRAY_SIMPLE_STRUCTURE_AUTO[2].WORD_TYPE + 1;

    ARRAY_SIMPLE_STRUCTURE_AUTO[3].BOOL_TYPE := NOT ARRAY_SIMPLE_STRUCTURE_AUTO[3].BOOL_TYPE;
    ARRAY_SIMPLE_STRUCTURE_AUTO[3].BYTE_TYPE := ARRAY_SIMPLE_STRUCTURE_AUTO[3].BYTE_TYPE + 1;
    ARRAY_SIMPLE_STRUCTURE_AUTO[3].DATE_TYPE := ANY_TO_DATE(1445385600 + ARRAY_SIMPLE_STRUCTURE_AUTO[3].DINT_TYPE * 86400);
    ARRAY_SIMPLE_STRUCTURE_AUTO[3].DINT_TYPE := ARRAY_SIMPLE_STRUCTURE_AUTO[3].DINT_TYPE + 1;
    ARRAY_SIMPLE_STRUCTURE_AUTO[3].DWORD_TYPE := ARRAY_SIMPLE_STRUCTURE_AUTO[3].DWORD_TYPE + 1;
    ARRAY_SIMPLE_STRUCTURE_AUTO[3].INT_TYPE := ARRAY_SIMPLE_STRUCTURE_AUTO[3].INT_TYPE + 1;
    ARRAY_SIMPLE_STRUCTURE_AUTO[3].LINT_TYPE := ARRAY_SIMPLE_STRUCTURE_AUTO[3].LINT_TYPE + 1;
    ARRAY_SIMPLE_STRUCTURE_AUTO[3].LREAL_TYPE := ARRAY_SIMPLE_STRUCTURE_AUTO[3].LREAL_TYPE + 1;
    ARRAY_SIMPLE_STRUCTURE_AUTO[3].LWORD_TYPE := ARRAY_SIMPLE_STRUCTURE_AUTO[3].LWORD_TYPE + 1;
    ARRAY_SIMPLE_STRUCTURE_AUTO[3].REAL_TYPE := ARRAY_SIMPLE_STRUCTURE_AUTO[3].REAL_TYPE + 1;
    ARRAY_SIMPLE_STRUCTURE_AUTO[3].SINT_TYPE := ARRAY_SIMPLE_STRUCTURE_AUTO[3].SINT_TYPE + 1;
    ARRAY_SIMPLE_STRUCTURE_AUTO[3].STRING_TYPE := ANY_TO_STRING(ARRAY_SIMPLE_STRUCTURE_AUTO[3].DINT_TYPE) + ' ' + ANY_TO_STRING(ARRAY_SIMPLE_STRUCTURE_AUTO[3].TIME_TYPE);
    ARRAY_SIMPLE_STRUCTURE_AUTO[3].TIME_TYPE := ARRAY_SIMPLE_STRUCTURE_AUTO[3].TIME_TYPE + PULSE_TIME;
    ARRAY_SIMPLE_STRUCTURE_AUTO[3].UDINT_TYPE := ARRAY_SIMPLE_STRUCTURE_AUTO[3].UDINT_TYPE + 1;
    ARRAY_SIMPLE_STRUCTURE_AUTO[3].UINT_TYPE := ARRAY_SIMPLE_STRUCTURE_AUTO[3].UINT_TYPE + 1;
    ARRAY_SIMPLE_STRUCTURE_AUTO[3].ULINT_TYPE := ARRAY_SIMPLE_STRUCTURE_AUTO[3].ULINT_TYPE + 1;
    ARRAY_SIMPLE_STRUCTURE_AUTO[3].USINT_TYPE := ARRAY_SIMPLE_STRUCTURE_AUTO[3].USINT_TYPE + 1;
    ARRAY_SIMPLE_STRUCTURE_AUTO[3].WORD_TYPE := ARRAY_SIMPLE_STRUCTURE_AUTO[3].WORD_TYPE + 1;

    ARRAY_SIMPLE_STRUCTURE_AUTO[4].BOOL_TYPE := NOT ARRAY_SIMPLE_STRUCTURE_AUTO[4].BOOL_TYPE;
    ARRAY_SIMPLE_STRUCTURE_AUTO[4].BYTE_TYPE := ARRAY_SIMPLE_STRUCTURE_AUTO[4].BYTE_TYPE + 1;
    ARRAY_SIMPLE_STRUCTURE_AUTO[4].DATE_TYPE := ANY_TO_DATE(1445385600 + ARRAY_SIMPLE_STRUCTURE_AUTO[4].DINT_TYPE * 86400);
    ARRAY_SIMPLE_STRUCTURE_AUTO[4].DINT_TYPE := ARRAY_SIMPLE_STRUCTURE_AUTO[4].DINT_TYPE + 1;
    ARRAY_SIMPLE_STRUCTURE_AUTO[4].DWORD_TYPE := ARRAY_SIMPLE_STRUCTURE_AUTO[4].DWORD_TYPE + 1;
    ARRAY_SIMPLE_STRUCTURE_AUTO[4].INT_TYPE := ARRAY_SIMPLE_STRUCTURE_AUTO[4].INT_TYPE + 1;
    ARRAY_SIMPLE_STRUCTURE_AUTO[4].LINT_TYPE := ARRAY_SIMPLE_STRUCTURE_AUTO[4].LINT_TYPE + 1;
    ARRAY_SIMPLE_STRUCTURE_AUTO[4].LREAL_TYPE := ARRAY_SIMPLE_STRUCTURE_AUTO[4].LREAL_TYPE + 1;
    ARRAY_SIMPLE_STRUCTURE_AUTO[4].LWORD_TYPE := ARRAY_SIMPLE_STRUCTURE_AUTO[4].LWORD_TYPE + 1;
    ARRAY_SIMPLE_STRUCTURE_AUTO[4].REAL_TYPE := ARRAY_SIMPLE_STRUCTURE_AUTO[4].REAL_TYPE + 1;
    ARRAY_SIMPLE_STRUCTURE_AUTO[4].SINT_TYPE := ARRAY_SIMPLE_STRUCTURE_AUTO[4].SINT_TYPE + 1;
    ARRAY_SIMPLE_STRUCTURE_AUTO[4].STRING_TYPE := ANY_TO_STRING(ARRAY_SIMPLE_STRUCTURE_AUTO[4].DINT_TYPE) + ' ' + ANY_TO_STRING(ARRAY_SIMPLE_STRUCTURE_AUTO[4].TIME_TYPE);
    ARRAY_SIMPLE_STRUCTURE_AUTO[4].TIME_TYPE := ARRAY_SIMPLE_STRUCTURE_AUTO[4].TIME_TYPE + PULSE_TIME;
    ARRAY_SIMPLE_STRUCTURE_AUTO[4].UDINT_TYPE := ARRAY_SIMPLE_STRUCTURE_AUTO[4].UDINT_TYPE + 1;
    ARRAY_SIMPLE_STRUCTURE_AUTO[4].UINT_TYPE := ARRAY_SIMPLE_STRUCTURE_AUTO[4].UINT_TYPE + 1;
    ARRAY_SIMPLE_STRUCTURE_AUTO[4].ULINT_TYPE := ARRAY_SIMPLE_STRUCTURE_AUTO[4].ULINT_TYPE + 1;
    ARRAY_SIMPLE_STRUCTURE_AUTO[4].USINT_TYPE := ARRAY_SIMPLE_STRUCTURE_AUTO[4].USINT_TYPE + 1;
    ARRAY_SIMPLE_STRUCTURE_AUTO[4].WORD_TYPE := ARRAY_SIMPLE_STRUCTURE_AUTO[4].WORD_TYPE + 1;

    ARRAY_SIMPLE_STRUCTURE_AUTO[5].BOOL_TYPE := ARRAY_SIMPLE_STRUCTURE_AUTO[4].BOOL_TYPE;
    ARRAY_SIMPLE_STRUCTURE_AUTO[5].BYTE_TYPE := ARRAY_SIMPLE_STRUCTURE_AUTO[4].BYTE_TYPE;
    ARRAY_SIMPLE_STRUCTURE_AUTO[5].DATE_TYPE := ARRAY_SIMPLE_STRUCTURE_AUTO[4].DATE_TYPE;
    ARRAY_SIMPLE_STRUCTURE_AUTO[5].DINT_TYPE := ARRAY_SIMPLE_STRUCTURE_AUTO[4].DINT_TYPE;
    ARRAY_SIMPLE_STRUCTURE_AUTO[5].DWORD_TYPE := ARRAY_SIMPLE_STRUCTURE_AUTO[4].DWORD_TYPE;
    ARRAY_SIMPLE_STRUCTURE_AUTO[5].INT_TYPE := ARRAY_SIMPLE_STRUCTURE_AUTO[4].INT_TYPE;
    ARRAY_SIMPLE_STRUCTURE_AUTO[5].LINT_TYPE := ARRAY_SIMPLE_STRUCTURE_AUTO[4].LINT_TYPE;
    ARRAY_SIMPLE_STRUCTURE_AUTO[5].LREAL_TYPE := ARRAY_SIMPLE_STRUCTURE_AUTO[4].LREAL_TYPE;
    ARRAY_SIMPLE_STRUCTURE_AUTO[5].LWORD_TYPE := ARRAY_SIMPLE_STRUCTURE_AUTO[4].LWORD_TYPE;
    ARRAY_SIMPLE_STRUCTURE_AUTO[5].REAL_TYPE := ARRAY_SIMPLE_STRUCTURE_AUTO[4].REAL_TYPE;
    ARRAY_SIMPLE_STRUCTURE_AUTO[5].SINT_TYPE := ARRAY_SIMPLE_STRUCTURE_AUTO[4].SINT_TYPE;
    ARRAY_SIMPLE_STRUCTURE_AUTO[5].STRING_TYPE := ARRAY_SIMPLE_STRUCTURE_AUTO[4].STRING_TYPE;
    ARRAY_SIMPLE_STRUCTURE_AUTO[5].TIME_TYPE := ARRAY_SIMPLE_STRUCTURE_AUTO[4].TIME_TYPE;
    ARRAY_SIMPLE_STRUCTURE_AUTO[5].UDINT_TYPE := ARRAY_SIMPLE_STRUCTURE_AUTO[4].UDINT_TYPE;
    ARRAY_SIMPLE_STRUCTURE_AUTO[5].UINT_TYPE := ARRAY_SIMPLE_STRUCTURE_AUTO[4].UINT_TYPE;
    ARRAY_SIMPLE_STRUCTURE_AUTO[5].ULINT_TYPE := ARRAY_SIMPLE_STRUCTURE_AUTO[4].ULINT_TYPE;
    ARRAY_SIMPLE_STRUCTURE_AUTO[5].USINT_TYPE := ARRAY_SIMPLE_STRUCTURE_AUTO[4].USINT_TYPE;
    ARRAY_SIMPLE_STRUCTURE_AUTO[5].WORD_TYPE := ARRAY_SIMPLE_STRUCTURE_AUTO[4].WORD_TYPE;

END_IF;

END_PROGRAM
